	REGION READ AND INIT
	    
	    REGION Init conveyor parameters
	        
	        // Conveyor Parameter
	        // ProductionLine
	        IF #Active.Line.ProductionLine THEN
	            #ReadTransferParameters := DB_ConveyorParameters.Line.ProductionLine.Conveyor[#TransferID];
	        END_IF;
	        // EmptyLine
	        IF #Active.Line.EmptyLine THEN
	            #ReadTransferParameters := DB_ConveyorParameters.Line.EmptyLine.Conveyor[#TransferID];
	        END_IF;
	        // PackedLine
	        IF #Active.Line.PackedLine THEN
	            #ReadTransferParameters := DB_ConveyorParameters.Line.PackedLine.Conveyor[#TransferID];
	        END_IF;
	        
	    END_REGION
	    
	    REGION Sensor Filter
	        
	        // FB_Sensor
	        // called as MIDB
	        
	        #TRANSFER_SENSOR(Sensor := #ReadInputSignal.TransferSensor,
	                         SensorFilterTime := #ReadTransferParameters.SensorFilterTime,
	                         FilteredSensor => #FilteredSensor);
	        
	        // front sensor filter
	        #FRONT_SENSOR_FILTER(Sensor := #FrontSensor,
	                             SensorFilterTime := #FrontSensorFilterTime);
	        
	    END_REGION
	    
	    REGION FIRE
	        
	        // Fire signal from fire system stops the whole system
	        // System can be reset from Fire status only if the fire signal is deactivated
	        
	        // FIRE ALARM ACTIVE --> STOP SYSTEM
	        IF #ReadInputSignal.FireActive THEN
	            #StopSystemFireActive := TRUE;
	        END_IF;
	        // RESET --> FIRE ALARM
	        IF #SSR.ResetSystem AND NOT #ReadInputSignal.FireActive THEN
	            #StopSystemFireActive := FALSE;
	        END_IF;
	        
	    END_REGION
	    
	END_REGION
	
	REGION Conveyor Status
	    
	    REGION Status ON
	        
	        // ----------------------------------------->>>>>>> STATUS ON <<<<<<<-----------------------------------------
	        // FB_ConveyorStatusON
	        // called as IDMB
	        
	        #TRANSFER_STATUS_ON(SystemStartActive := #SSR.StartSystem,
	                            StatusStop := #ReadTransferStatus.Stop,
	                            StatusEStop := #ReadTransferStatus.Estop,
	                            StatusManual := #ReadTransferStatus.Manual,
	                            StatusFault := #ReadTransferStatus.Fault,
	                            FireAlarmActive := #StopSystemFireActive,
	                            StatusON => #ReadTransferStatus.ON);
	        
	    END_REGION
	    
	    REGION Status Ready
	        
	        // ----------------------------------------->>>>>>> STATUS READY <<<<<<<-----------------------------------------
	        // FB_ConveyorStatusReady
	        // called as MIDB
	        
	        #TRANSFER_STATUS_READY(StatusON := #ReadTransferStatus.ON,
	                               StatusESTOP := #ReadTransferStatus.Estop,
	                               StatusFAULT := #ReadTransferStatus.Fault,
	                               StatusMAN := #ReadTransferStatus.Manual,
	                               SignalFIRE := #StopSystemFireActive,
	                               SystemAlertTime := #ReadTransferParameters.StartUpTime,
	                               StatusReady => #ReadTransferStatus.ReadytoRun);
	        
	    END_REGION
	    
	    REGION Status Occupied
	        
	        // ----------------------------------------->>>>>>> STATUS OCCUPIED <<<<<<<-----------------------------------------
	        
	        #ReadTransferStatus.Occupied :=
	        #FilteredSensor AND
	        NOT #FRONT_SENSOR_FILTER.FilteredSensor;
	        
	    END_REGION
	    
	    REGION Status Running
	        
	        // ----------------------------------------->>>>>>> STATUS RUNNING <<<<<<<-----------------------------------------
	        
	        #ReadTransferStatus.Running := #Transfer.Command_1 OR #Transfer.Command_2;
	        
	    END_REGION
	    
	    REGION Status Fault
	        
	        // Automatic reset trigger to the needed drive after wakeup from ESTOP power miss (only if needed)
	        // will trigger for every Reset active
	        
	        #AUTO_RESET(AckIN := #SSR.ResetSystem,
	                    Ack => #AutoReset);
	        
	        // ----------------------------------------->>>>>>> STATUS FAULT <<<<<<<-----------------------------------------
	        // FC_ConveyorStatusFault
	        #TRANSFER_STATUS_FAULT(FaultActive := #ReadInputSignal.Fault,
	                               ResetFault := #SSR.ResetSystem OR #AutoReset,
	                               StatusRunning := #ReadTransferStatus.Running,
	                               FaultStatus => #ReadTransferStatus.Fault);
	        
	        #ErrorReset := #SSR.ResetSystem;
	        
	    END_REGION
	    
	    REGION Status ESTOP
	        
	        // ----------------------------------------->>>>>>> STATUS ESTOP <<<<<<<-----------------------------------------
	        
	        // EMERGENCY STOP ACTIVE --> STOP SYSTEM
	        IF #ReadInputSignal.EmergencyStop THEN
	            #ReadTransferStatus.Estop := TRUE;
	        END_IF;
	        // RESET --> EMERGENCY STOP
	        IF #AutoReset AND NOT #ReadInputSignal.EmergencyStop THEN
	            #ReadTransferStatus.Estop := FALSE;
	        END_IF;
	        
	    END_REGION
	    
	    REGION Status Manual
	        
	        // ----------------------------------------->>>>>>> STATUS MANUAL <<<<<<<-----------------------------------------
	        
	        // Write to static from IO
	        // ACTIVATE --> MANUAL MODE
	        // ProductionLine
	        IF #Active.Line.ProductionLine THEN
	            // SET --> MANUAL MODE
	            IF DB_Manual.Line.ProductionLine.Conveyor[#TransferID].ManualEnable THEN
	                #ReadTransferStatus.Manual := TRUE;
	            END_IF;
	            // RESET --> MANUAL MODE
	            IF NOT DB_Manual.Line.ProductionLine.Conveyor[#TransferID].ManualEnable AND #SSR.ResetSystem THEN
	                #ReadTransferStatus.Manual := FALSE;
	            END_IF;
	        END_IF;
	        // EmptyLine
	        IF #Active.Line.EmptyLine THEN
	            // SET --> MANUAL MODE
	            IF DB_Manual.Line.EmptyLine.Conveyor[#TransferID].ManualEnable THEN
	                #ReadTransferStatus.Manual := TRUE;
	            END_IF;
	            // RESET --> MANUAL MODE
	            IF NOT DB_Manual.Line.EmptyLine.Conveyor[#TransferID].ManualEnable AND #SSR.ResetSystem THEN
	                #ReadTransferStatus.Manual := FALSE;
	            END_IF;
	        END_IF;
	        // PackedLine
	        IF #Active.Line.PackedLine THEN
	            // SET --> MANUAL MODE
	            IF DB_Manual.Line.PackedLine.Conveyor[#TransferID].ManualEnable THEN
	                #ReadTransferStatus.Manual := TRUE;
	            END_IF;
	            // RESET --> MANUAL MODE
	            IF NOT DB_Manual.Line.PackedLine.Conveyor[#TransferID].ManualEnable AND #SSR.ResetSystem THEN
	                #ReadTransferStatus.Manual := FALSE;
	            END_IF;
	        END_IF;
	        
	    END_REGION
	    
	    REGION Status Stop
	        
	        // ----------------------------------------->>>>>>> STATUS STOP <<<<<<<-----------------------------------------
	        
	        IF #SSR.StopSystem THEN
	            #ReadTransferStatus.Stop := TRUE;
	        END_IF;
	        IF #SSR.StartSystem OR #SSR.ResetSystem THEN
	            #ReadTransferStatus.Stop := FALSE;
	        END_IF;
	        
	    END_REGION
	    
	    REGION Status Blockage
	        
	        // FB_SensorBlockage
	        // called as MIDB
	        #TRANSFER_SENSOR_BLOCKAGE(IN := #ReadTransferStatus.ReadytoRun AND #FilteredSensor AND NOT #Downstream,
	                                  PT := T#15s);
	        
	        #FRONT_SENSOR_BLOCKAGE(IN := #ReadTransferStatus.ReadytoRun AND #FrontSensor AND NOT #Downstream,
	                               PT := T#15s);
	        
	        #END_SENSOR_BLOCKAGE(IN := #ReadTransferStatus.ReadytoRun AND #EndSensor AND NOT #Downstream,
	                             PT := T#15s);
	        
	        #"LEFT/RIGHT_SENSOR_BLOCKAGE"(IN := #ReadTransferStatus.ReadytoRun AND #"Left/RightSensor" AND NOT #Downstream,
	                                      PT := T#5s);
	        
	        #ReadTransferStatus.Blockage :=
	        (#TRANSFER_SENSOR_BLOCKAGE.Q OR
	        #FRONT_SENSOR_BLOCKAGE.Q OR
	        #END_SENSOR_BLOCKAGE.Q OR
	        #"LEFT/RIGHT_SENSOR_BLOCKAGE".Q) AND
	        (#TransferDirection.Straight OR
	        #TransferDirection.toRight OR
	        #TransferDirection.toLeft);
	        
	        // ==========================
	        // Sensor Blockage: HMI Alarm
	        // ==========================
	        // Sensor blockage alarm message is written to the alarm word
	        // corresponding to the active line
	        
	        REGION alarm 
	            
	            // ==========================
	            // Sensor Blockage: HMI Alarm
	            // ==========================
	            // Sensor blockage alarm message is written to the alarm word
	            // corresponding to the active line
	            // ProductionLine
	            IF #Active.Line.ProductionLine THEN
	                DB_Alarm."word".Line.ProductionLine.Conveyor[#TransferID].%X0 := #ReadTransferStatus.Blockage;
	            END_IF;
	            // EmptyLine
	            IF #Active.Line.EmptyLine THEN
	                DB_Alarm."word".Line.EmptyLine.Conveyor[#TransferID].%X0 := #ReadTransferStatus.Blockage;
	            END_IF;
	            // PackedLine
	            IF #Active.Line.PackedLine THEN
	                DB_Alarm."word".Line.PackedLine.Conveyor[#TransferID].%X0 := #ReadTransferStatus.Blockage;
	            END_IF;
	            
	        END_REGION
	        
	    END_REGION
	    
	    REGION Visu Color
	        
	        // each and every status of the conveyor will be mentioned by different colors in HMI panel
	        
	        #VisuColor.%X8 := #ReadTransferStatus.Blockage;
	        #VisuColor.%X0 := #ReadTransferStatus.ON;
	        #VisuColor.%X1 := #ReadTransferStatus.ReadytoRun;
	        #VisuColor.%X2 := #ReadTransferStatus.Occupied;
	        #VisuColor.%X3 := #ReadTransferStatus.Running;
	        #VisuColor.%X4 := #ReadTransferStatus.Fault;
	        #VisuColor.%X5 := #ReadTransferStatus.Estop;
	        #VisuColor.%X6 := #ReadTransferStatus.Manual;
	        #VisuColor.%X7 := #ReadTransferStatus.Stop;
	        
	        // convert word to Interger value: 
	        // color will be depends on the status priority (integer value) 
	        // reference: Conveyor image in HMI screen -> property -> Apperance   
	        
	        // ProductionLine
	        IF #Active.Line.ProductionLine THEN
	            DB_VisuColor.Line.ProductionLine.Conveyor[#TransferID] :=
	            WORD_TO_INT(#VisuColor);
	        END_IF;
	        // EmptyLine
	        IF #Active.Line.EmptyLine THEN
	            DB_VisuColor.Line.EmptyLine.Conveyor[#TransferID] :=
	            WORD_TO_INT(#VisuColor);
	        END_IF;
	        // PackedLine
	        IF #Active.Line.PackedLine THEN
	            DB_VisuColor.Line.PackedLine.Conveyor[#TransferID] :=
	            WORD_TO_INT(#VisuColor);
	        END_IF;
	        
	    END_REGION
	    
	    REGION Global Status
	        
	        // write -> global status
	        // ProductionLine
	        IF #Active.Line.ProductionLine THEN
	            DB_Global.Status.Line.ProductionLine.On[#TransferID] := #ReadTransferStatus.ON;
	            DB_Global.Status.Line.ProductionLine.ReadyToRun[#TransferID] := #ReadTransferStatus.ReadytoRun;
	            DB_Global.Status.Line.ProductionLine.Occupied[#TransferID] := #ReadTransferStatus.Occupied;
	            DB_Global.Status.Line.ProductionLine.Running[#TransferID] := #ReadTransferStatus.Running;
	            DB_Global.Status.Line.ProductionLine.Fault[#TransferID] := #ReadTransferStatus.Fault;
	            DB_Global.Status.Line.ProductionLine.Estop[#TransferID] := #ReadTransferStatus.Estop;
	            DB_Global.Status.Line.ProductionLine.Manual[#TransferID] := #ReadTransferStatus.Manual;
	            DB_Global.Status.Line.ProductionLine.Stop[#TransferID] := #ReadTransferStatus.Stop;
	            DB_Global.Status.Line.ProductionLine.Blockage[#TransferID] := #ReadTransferStatus.Blockage;
	        END_IF;
	        // EmptyLine
	        IF #Active.Line.EmptyLine THEN
	            DB_Global.Status.Line.EmptyLine.On[#TransferID] := #ReadTransferStatus.ON;
	            DB_Global.Status.Line.EmptyLine.ReadyToRun[#TransferID] := #ReadTransferStatus.ReadytoRun;
	            DB_Global.Status.Line.EmptyLine.Occupied[#TransferID] := #ReadTransferStatus.Occupied;
	            DB_Global.Status.Line.EmptyLine.Running[#TransferID] := #ReadTransferStatus.Running;
	            DB_Global.Status.Line.EmptyLine.Fault[#TransferID] := #ReadTransferStatus.Fault;
	            DB_Global.Status.Line.EmptyLine.Estop[#TransferID] := #ReadTransferStatus.Estop;
	            DB_Global.Status.Line.EmptyLine.Manual[#TransferID] := #ReadTransferStatus.Manual;
	            DB_Global.Status.Line.EmptyLine.Stop[#TransferID] := #ReadTransferStatus.Stop;
	            DB_Global.Status.Line.EmptyLine.Blockage[#TransferID] := #ReadTransferStatus.Blockage;
	        END_IF;
	        // PackedLine
	        IF #Active.Line.PackedLine THEN
	            DB_Global.Status.Line.PackedLine.On[#TransferID] := #ReadTransferStatus.ON;
	            DB_Global.Status.Line.PackedLine.ReadyToRun[#TransferID] := #ReadTransferStatus.ReadytoRun;
	            DB_Global.Status.Line.PackedLine.Occupied[#TransferID] := #ReadTransferStatus.Occupied;
	            DB_Global.Status.Line.PackedLine.Running[#TransferID] := #ReadTransferStatus.Running;
	            DB_Global.Status.Line.PackedLine.Fault[#TransferID] := #ReadTransferStatus.Fault;
	            DB_Global.Status.Line.PackedLine.Estop[#TransferID] := #ReadTransferStatus.Estop;
	            DB_Global.Status.Line.PackedLine.Manual[#TransferID] := #ReadTransferStatus.Manual;
	            DB_Global.Status.Line.PackedLine.Stop[#TransferID] := #ReadTransferStatus.Stop;
	            DB_Global.Status.Line.PackedLine.Blockage[#TransferID] := #ReadTransferStatus.Blockage;
	        END_IF;
	        
	    END_REGION
	    
	END_REGION
	
	REGION Transfer Logic
	    
	    REGION infeed receive condition
	        
	        // NegEdgeUpstream
	        #NegEdgeUpstream(CLK := #Upstream);
	        
	        // item will be send into the transfer section when there is no other item
	        
	        IF #ReadTransferStatus.ReadytoRun AND
	            #Upstream AND
	            NOT #ReadTransferStatus.Occupied THEN
	            #Transfer.RcvInfeed := TRUE;
	        END_IF;
	        
	        // receive infeed tag goes to FALSE when the item from the previous conveyor is completly out of the previous conveyor
	        IF NOT #Upstream(* #NegEdgeUpstream.Q *)THEN
	            #Transfer.RcvInfeed := FALSE;
	        END_IF;
	        
	        // Receive infeed
	        #Transfer.StartSignal := #Transfer.RcvInfeed;
	        
	    END_REGION
	    
	    REGION Transfer direction outputs
	        
	        IF NOT #EndSensor AND NOT #"Left/RightSensor" AND NOT #ReadTransferStatus.Running THEN
	            
	            #sTransferDirection := #TransferDirection;
	            
	        END_IF;
	        
	        // Transfer Straight
	        
	        IF #sTransferDirection.Straight THEN
	            
	            IF #ReadTransferStatus.ReadytoRun AND
	                NOT #Transfer.RcvInfeed AND
	                #ReadTransferStatus.Occupied AND
	                NOT #Downstream
	            THEN
	                #Transfer.Command_1 := TRUE;
	                #Transfer.Command_2 := TRUE;
	            END_IF;
	            
	        END_IF;
	        
	        // Transfer Right
	        
	        IF #sTransferDirection.toRight THEN
	            
	            IF #ReadTransferStatus.ReadytoRun AND
	                NOT #Transfer.RcvInfeed AND
	                #ReadTransferStatus.Occupied AND
	                NOT #Downstream
	            THEN
	                #Transfer.Command_1 := TRUE;
	                #Transfer.Command_2 := FALSE;
	            END_IF;
	            
	        END_IF;
	        
	        // Transfer Left
	        
	        IF #sTransferDirection.toLeft THEN
	            
	            IF #ReadTransferStatus.ReadytoRun AND
	                NOT #Transfer.RcvInfeed AND
	                #ReadTransferStatus.Occupied AND
	                NOT #Downstream
	            THEN
	                #Transfer.Command_1 := FALSE;
	                #Transfer.Command_2 := TRUE;
	            END_IF;
	            
	        END_IF;
	        
	    END_REGION
	    
	    REGION TRANSFER OFF
	        
	        // Transfer commands Off
	        
	        IF NOT #ReadTransferStatus.ReadytoRun OR
	            #Transfer.RcvInfeed OR
	            (#ReadTransferStatus.Occupied AND
	            #Downstream) OR
	            NOT #ReadTransferStatus.Occupied
	        THEN
	            #Transfer.Command_1 := FALSE;
	            #Transfer.Command_2 := FALSE;
	        END_IF;
	        
	    END_REGION
	    
	    REGION Write output
	        
	        // Static to output
	        
	        #StartSignal := #Transfer.StartSignal;
	        #Cmd1 := #Transfer.Command_1;
	        #Cmd2 := #Transfer.Command_2;
	        
	    END_REGION
	    
	END_REGION
	
	
	
	
	
END_FUNCTION_BLOCK
END_NAMESPACE

NAMESPACE Global
FUNCTION_BLOCK FB_GetDiag
{ S7_Optimized_Access := 'TRUE' ; Published := 'TRUE' }
VERSION : 0.1
   VAR_INPUT 
      HardwareID : HW_ANY;
   END_VAR

   VAR_OUTPUT 
      CommunicationErrorAlarm : Bool;
   END_VAR

   VAR 
      GetDiag { S7_SetPoint := 'False'} : GetDiag;
      CheckOwnState : UInt := 5;
      CommunicationError : Bool;
   END_VAR


BEGIN
	// ==========================================================================================================================================
	// Company        : LogTech, s.r.o.
	// Created by     : Anton Vinoth Soundraraj
	// Block          : FB_GetDiag
	// Project        : LT-Lib-Block
	// ==========================================================================================================================================
	
	REGION Get_Diag
	    
	    #GetDiag.ReturnValue := GET_DIAG(MODE := #GetDiag.DiagMode,
	                                     LADDR := #HardwareID,
	                                     CNT_DIAG => #GetDiag.CountDiagDetail,
	                                     DIAG := #GetDiag.MyDiag);
	END_REGION
	
	REGION Communiation_Error
	    
	    IF #GetDiag.MyDiag.OwnState = #CheckOwnState THEN
	        #CommunicationErrorAlarm := TRUE;
	    ELSE
	        #CommunicationErrorAlarm := FALSE;
	    END_IF;
	    
	    IF #GetDiag.MyDiag.OwnState = #CheckOwnState THEN
	        #CommunicationError := TRUE;
	    ELSE
	        #CommunicationError := FALSE;
	    END_IF;
	    
	END_REGION
	
	
END_FUNCTION_BLOCK
END_NAMESPACE

NAMESPACE Global
FUNCTION_BLOCK FB_HardwareDiag
{ S7_Optimized_Access := 'TRUE' ; Published := 'TRUE' }
VERSION : 0.1
   VAR 
      "BW-ASi -10.106.129.143" { S7_SetPoint := 'False'} : FB_GetDiag;
      "BW-ASi -10.106.129.200" : FB_GetDiag;
      "Cognex -10.106.129.24" { S7_SetPoint := 'False'} : FB_GetDiag;
      "Cognex -10.106.129.25" : FB_GetDiag;
      "Cognex -10.106.129.26" : FB_GetDiag;
      "Cognex -10.106.129.27" : FB_GetDiag;
      "IMC - 10.106.129.84" : FB_GetDiag;
      "IMC - 10.106.129.85" : FB_GetDiag;
      "IMC - 10.106.129.86" : FB_GetDiag;
      "IMC - 10.106.129.87" : FB_GetDiag;
      "IMC - 10.106.129.88" : FB_GetDiag;
   END_VAR


BEGIN
	// ==========================================================================================================================================
	// Company        : LogTech, s.r.o.
	// Created by     : Anton Vinoth Soundraraj
	// Block          : FB_HardwareDiag
	// Project        : Lékarna DC Chrudim
	// Project number : 23-157
	// ==========================================================================================================================================
	
	
	REGION BW ASi module
	    
	    
	    #"BW-ASi -10.106.129.143"(CommunicationErrorAlarm=> DB_Alarm.CommunicationFault."BW-ASi".%X0);  // remove for simulation testing HardwareID:= _."ASi-GW~IODevice",
	    
	    #"BW-ASi -10.106.129.200"(CommunicationErrorAlarm=> DB_Alarm.CommunicationFault."BW-ASi".%X1);
	    
	END_REGION
	
	
	REGION Cognex
	    
	    #"Cognex -10.106.129.24"(CommunicationErrorAlarm=> DB_Alarm.CommunicationFault.Cognex.%X0);
	    
	    
	    #"Cognex -10.106.129.25"(CommunicationErrorAlarm=> DB_Alarm.CommunicationFault.Cognex.%X1);
	    
	    
	    #"Cognex -10.106.129.26"(CommunicationErrorAlarm=> DB_Alarm.CommunicationFault.Cognex.%X2);
	    
	    
	    #"Cognex -10.106.129.27"(CommunicationErrorAlarm=> DB_Alarm.CommunicationFault.Cognex.%X3);
	    
	    
	END_REGION
	
	REGION IMC
	    
	    #"IMC - 10.106.129.84"(CommunicationErrorAlarm=>DB_Alarm.CommunicationFault.IMC.%X0);
	    
	    #"IMC - 10.106.129.85"(CommunicationErrorAlarm=>DB_Alarm.CommunicationFault.IMC.%X1);
	    
	    #"IMC - 10.106.129.86"(CommunicationErrorAlarm=>DB_Alarm.CommunicationFault.IMC.%X1);
	    
	    #"IMC - 10.106.129.87"(CommunicationErrorAlarm=>DB_Alarm.CommunicationFault.IMC.%X2);
	    
	    #"IMC - 10.106.129.88"(CommunicationErrorAlarm=>DB_Alarm.CommunicationFault.IMC.%X3);
	    
	END_REGION
	
	
	
	
	
	
	
END_FUNCTION_BLOCK
END_NAMESPACE

NAMESPACE Global
FUNCTION_BLOCK FB_VisuAlarm
{ S7_Optimized_Access := 'TRUE' ; Published := 'TRUE' }
VERSION : 0.1
   VAR 
      noAlarmState : Bool;
      CommunicationFault : Struct
         PLC : Word;
         "BW-ASi" : Word;
         Cognex : Word;
         Mabs : Word;
      END_STRUCT;
      "BW-ASi" : Struct
         "BW_ASi143 -MCC100 -210KE3 -ConfigErr_Circuit1_Slave(0-15)A_1" : Word;
         "BW_ASi143 -MCC100 -210KE3 -ConfigErr_Circuit1_Slave(16-31)A" : Word;
         "BW_ASi143 -MCC100 -210KE3 -ConfigErr_Circuit1_Slave(0-15)B_1" : Word;
         "BW_ASi143 -MCC100 -210KE3 -ConfigErr_Circuit1_Slave(16-31)B" : Word;
         "BW_ASi143 -MCC100 -210KE3 -PeriErr_Circuit1_Slave(0-15)A_1" : Word;
         "BW_ASi143 -MCC100 -210KE3 -PeriErr_Circuit1_Slave(16-31)A" : Word;
         "BW_ASi143 -MCC100 -210KE3 -PeriErr_Circuit1_Slave(0-15)B_1" : Word;
         "BW_ASi143 -MCC100 -210KE3 -PeriErr_Circuit1_Slave(16-31)B" : Word;
         "BW_ASi143 -MCC100 -210KE3 -ConfigErr_Circuit2_Slave(0-15)A" : Word;
         "BW_ASi143 -MCC100 -210KE3 -ConfigErr_Circuit2_Slave(16-31)A" : Word;
         "BW_ASi143 -MCC100 -210KE3 -ConfigErr_Circuit2_Slave(0-15)B" : Word;
         "BW_ASi143 -MCC100 -210KE3 -ConfigErr_Circuit2_Slave(16-31)B" : Word;
         "BW_ASi143 -MCC100 -210KE3 -PeriErr_Circuit2_Slave(0-15)A" : Word;
         "BW_ASi143 -MCC100 -210KE3 -PeriErr_Circuit2_Slave(16-31)A" : Word;
         "BW_ASi143 -MCC100 -210KE3 -PeriErr_Circuit2_Slave(0-15)B" : Word;
         "BW_ASi143 -MCC100 -210KE3 -PeriErr_Circuit2_Slave(16-31)B" : Word;
         "BW_ASi200 -MCC300 -210KE3 -ConfigErr_Circuit1_Slave(0-15)A" : Word;
         "BW_ASi200 -MCC300 -210KE3 -ConfigErr_Circuit1_Slave(16-31)A" : Word;
         "BW_ASi200 -MCC300 -210KE3 -ConfigErr_Circuit1_Slave(0-15)B" : Word;
         "BW_ASi200 -MCC300 -210KE3 -ConfigErr_Circuit1_Slave(16-31)B" : Word;
         "BW_ASi200 -MCC300 -210KE3 -PeriErr_Circuit1_Slave(0-15)A" : Word;
         "BW_ASi200 -MCC300 -210KE3 -PeriErr_Circuit1_Slave(16-31)A" : Word;
         "BW_ASi200 -MCC300 -210KE3 -PeriErr_Circuit1_Slave(0-15)B" : Word;
         "BW_ASi200 -MCC300 -210KE3 -PeriErr_Circuit1_Slave(16-31)B" : Word;
         "BW_ASi200 -MCC300 -210KE3 -ConfigErr_Circuit2_Slave(0-15)A" : Word;
         "BW_ASi200 -MCC300 -210KE3 -ConfigErr_Circuit2_Slave(16-31)A" : Word;
         "BW_ASi200 -MCC300 -210KE3 -ConfigErr_Circuit2_Slave(0-15)B" : Word;
         "BW_ASi200 -MCC300 -210KE3 -ConfigErr_Circuit2_Slave(16-31)B" : Word;
         "BW_ASi200 -MCC300 -210KE3 -PeriErr_Circuit2_Slave(0-15)A" : Word;
         "BW_ASi200 -MCC300 -210KE3 -PeriErr_Circuit2_Slave(16-31)A" : Word;
         "BW_ASi200 -MCC300 -210KE3 -PeriErr_Circuit2_Slave(0-15)B" : Word;
         "BW_ASi200 -MCC300 -210KE3 -PeriErr_Circuit2_Slave(16-31)B" : Word;
      END_STRUCT;
      "word" : Struct
         Line : Struct
            ProductionLine : Struct
               Conveyor : Array[_.gminProductionLine.._.gmaxProductionLine] of Word;
            END_STRUCT;
            EmptyLine : Struct
               Conveyor : Array[_.gminEmptyLine.._.gmaxEmptyLine] of Word;
            END_STRUCT;
            PackedLine : Struct
               Conveyor : Array[_.gminPackedLine.._.gmaxPackedLine] of Word;
            END_STRUCT;
         END_STRUCT;
      END_STRUCT;
   END_VAR


BEGIN
	// ==========================================================================================================================================
	// Company        : LogTech, s.r.o.
	// Created by     : Mahmoud Elnady
	// Block          : FC_VisuAlarm
	// Project        : Lékárna Chrudim
	// Project number : 23-157
	// ==========================================================================================================================================
	REGION initial state
	    
	    // ESTOP alarm has priority
	    // So, if there are any estop active, other alarms can't be displayed on Alarm screen
	    
	    // no alarm state
	    #noAlarmState :=
	    IDB_GlobalStatus.Line.ProductionLine.Estop OR
	    IDB_GlobalStatus.Line.ProductionLine.Estop OR
	    IDB_GlobalStatus.Line.ProductionLine.Estop;
	    
	    IF #noAlarmState THEN
	        
	        DB_Alarm."BW-ASi" := #"BW-ASi";
	        DB_Alarm.CommunicationFault := #CommunicationFault;
	        DB_Alarm."word" := #word;
	        //"DB_Alarm".CircuitBreaker := #CircuitBreaker;
	        
	    END_IF;
	    
	END_REGION
	
	REGION ASi Config and Peri alarm
	    
	    IF NOT #noAlarmState THEN
	        // ASi gateway: MCC100-bw23: Circuit 1
	        DB_Alarm."BW-ASi"."BW_ASi143 -MCC100 -210KE3 -ConfigErr_Circuit1_Slave(0-15)A" := _."BW_ASi143 -MCC100 -210KE3 -ConfigErr_Circuit1_Slave(0-15)A";
	        DB_Alarm."BW-ASi"."BW_ASi143 -MCC100 -210KE3 -ConfigErr_Circuit1_Slave(16-31)A" := _."BW_ASi143 -MCC100 -210KE3 -ConfigErr_Circuit1_Slave(16-31)A";
	        DB_Alarm."BW-ASi"."BW_ASi143 -MCC100 -210KE3 -ConfigErr_Circuit1_Slave(0-15)B" := _."BW_ASi143 -MCC100 -210KE3 -ConfigErr_Circuit1_Slave(0-15)B";
	        DB_Alarm."BW-ASi"."BW_ASi143 -MCC100 -210KE3 -ConfigErr_Circuit1_Slave(16-31)B" := _."BW_ASi143 -MCC100 -210KE3 -ConfigErr_Circuit1_Slave(16-31)B";
	        DB_Alarm."BW-ASi"."BW_ASi143 -MCC100 -210KE3 -PeriErr_Circuit1_Slave(0-15)A" := _."BW_ASi143 -MCC100 -210KE3 -PeriErr_Circuit1_Slave(0-15)A";
	        DB_Alarm."BW-ASi"."BW_ASi143 -MCC100 -210KE3 -PeriErr_Circuit1_Slave(16-31)A" := _."BW_ASi143 -MCC100 -210KE3 -PeriErr_Circuit1_Slave(16-31)A";
	        DB_Alarm."BW-ASi"."BW_ASi143 -MCC100 -210KE3 -PeriErr_Circuit1_Slave(0-15)B" := _."BW_ASi143 -MCC100 -210KE3 -PeriErr_Circuit1_Slave(0-15)B";
	        DB_Alarm."BW-ASi"."BW_ASi143 -MCC100 -210KE3 -PeriErr_Circuit1_Slave(16-31)B" := _."BW_ASi143 -MCC100 -210KE3 -PeriErr_Circuit1_Slave(16-31)B";
	        // ASi gateway: MCC100-bw23: Circuit 2
	        DB_Alarm."BW-ASi"."BW_ASi143 -MCC100 -210KE3 -ConfigErr_Circuit1_Slave(0-15)A" := _."BW_ASi143 -MCC100 -210KE3 -ConfigErr_Circuit1_Slave(0-15)A";
	        DB_Alarm."BW-ASi"."BW_ASi143 -MCC100 -210KE3 -ConfigErr_Circuit1_Slave(16-31)A" := _."BW_ASi143 -MCC100 -210KE3 -ConfigErr_Circuit1_Slave(16-31)A";
	        DB_Alarm."BW-ASi"."BW_ASi143 -MCC100 -210KE3 -ConfigErr_Circuit1_Slave(0-15)B" := _."BW_ASi143 -MCC100 -210KE3 -ConfigErr_Circuit1_Slave(0-15)B";
	        DB_Alarm."BW-ASi"."BW_ASi143 -MCC100 -210KE3 -ConfigErr_Circuit1_Slave(16-31)B" := _."BW_ASi143 -MCC100 -210KE3 -ConfigErr_Circuit1_Slave(16-31)B";
	        DB_Alarm."BW-ASi"."BW_ASi143 -MCC100 -210KE3 -PeriErr_Circuit1_Slave(0-15)A" := _."BW_ASi143 -MCC100 -210KE3 -PeriErr_Circuit1_Slave(0-15)A";
	        DB_Alarm."BW-ASi"."BW_ASi143 -MCC100 -210KE3 -PeriErr_Circuit1_Slave(16-31)A" := _."BW_ASi143 -MCC100 -210KE3 -PeriErr_Circuit1_Slave(16-31)A";
	        DB_Alarm."BW-ASi"."BW_ASi143 -MCC100 -210KE3 -PeriErr_Circuit1_Slave(0-15)B" := _."BW_ASi143 -MCC100 -210KE3 -PeriErr_Circuit1_Slave(0-15)B";
	        DB_Alarm."BW-ASi"."BW_ASi143 -MCC100 -210KE3 -PeriErr_Circuit1_Slave(16-31)B" := _."BW_ASi143 -MCC100 -210KE3 -PeriErr_Circuit1_Slave(16-31)B";
	        // ASi gateway: MCC300-bw31 : Circuit 1
	        DB_Alarm."BW-ASi"."BW_ASi200 -MCC300 -210KE3 -ConfigErr_Circuit1_Slave(0-15)A" := _."BW_ASi200 -MCC300 -210KE3 -ConfigErr_Circuit1_Slave(0-15)A";
	        DB_Alarm."BW-ASi"."BW_ASi200 -MCC300 -210KE3 -ConfigErr_Circuit1_Slave(16-31)A" := _."BW_ASi200 -MCC300 -210KE3 -ConfigErr_Circuit1_Slave(16-31)A";
	        DB_Alarm."BW-ASi"."BW_ASi200 -MCC300 -210KE3 -ConfigErr_Circuit1_Slave(0-15)B" := _."BW_ASi200 -MCC300 -210KE3 -ConfigErr_Circuit1_Slave(0-15)B";
	        DB_Alarm."BW-ASi"."BW_ASi200 -MCC300 -210KE3 -ConfigErr_Circuit1_Slave(16-31)B" := _."BW_ASi200 -MCC300 -210KE3 -ConfigErr_Circuit1_Slave(16-31)B";
	        DB_Alarm."BW-ASi"."BW_ASi200 -MCC300 -210KE3 -PeriErr_Circuit1_Slave(0-15)A" := _."BW_ASi200 -MCC300 -210KE3 -PeriErr_Circuit1_Slave(0-15)A";
	        DB_Alarm."BW-ASi"."BW_ASi200 -MCC300 -210KE3 -PeriErr_Circuit1_Slave(16-31)A" := _."BW_ASi200 -MCC300 -210KE3 -PeriErr_Circuit1_Slave(16-31)A";
	        DB_Alarm."BW-ASi"."BW_ASi200 -MCC300 -210KE3 -PeriErr_Circuit1_Slave(0-15)B" := _."BW_ASi200 -MCC300 -210KE3 -PeriErr_Circuit1_Slave(0-15)B";
	        DB_Alarm."BW-ASi"."BW_ASi200 -MCC300 -210KE3 -PeriErr_Circuit1_Slave(16-31)B" := _."BW_ASi200 -MCC300 -210KE3 -PeriErr_Circuit1_Slave(16-31)B";
	        // ASi gateway: MCC300-bw31 : Circuit 2
	        DB_Alarm."BW-ASi"."BW_ASi200 -MCC300 -210KE3 -ConfigErr_Circuit2_Slave(0-15)A" := _."BW_ASi200 -MCC300 -210KE3 -ConfigErr_Circuit2_Slave(0-15)A";
	        DB_Alarm."BW-ASi"."BW_ASi200 -MCC300 -210KE3 -ConfigErr_Circuit2_Slave(16-31)A" := _."BW_ASi200 -MCC300 -210KE3 -ConfigErr_Circuit2_Slave(16-31)A";
	        DB_Alarm."BW-ASi"."BW_ASi200 -MCC300 -210KE3 -ConfigErr_Circuit2_Slave(0-15)B" := _."BW_ASi200 -MCC300 -210KE3 -ConfigErr_Circuit2_Slave(0-15)B";
	        DB_Alarm."BW-ASi"."BW_ASi200 -MCC300 -210KE3 -ConfigErr_Circuit2_Slave(16-31)B" := _."BW_ASi200 -MCC300 -210KE3 -ConfigErr_Circuit2_Slave(16-31)B";
	        DB_Alarm."BW-ASi"."BW_ASi200 -MCC300 -210KE3 -PeriErr_Circuit2_Slave(0-15)A" := _."BW_ASi200 -MCC300 -210KE3 -PeriErr_Circuit2_Slave(0-15)A";
	        DB_Alarm."BW-ASi"."BW_ASi200 -MCC300 -210KE3 -PeriErr_Circuit2_Slave(16-31)A" := _."BW_ASi200 -MCC300 -210KE3 -PeriErr_Circuit2_Slave(16-31)A";
	        DB_Alarm."BW-ASi"."BW_ASi200 -MCC300 -210KE3 -PeriErr_Circuit2_Slave(0-15)B" := _."BW_ASi200 -MCC300 -210KE3 -PeriErr_Circuit2_Slave(0-15)B";
	        DB_Alarm."BW-ASi"."BW_ASi200 -MCC300 -210KE3 -PeriErr_Circuit2_Slave(16-31)B" := _."BW_ASi200 -MCC300 -210KE3 -PeriErr_Circuit2_Slave(16-31)B";
	    ELSE
	        // ASi gateway: MCC100-bw23: Circuit 1
	        DB_Alarm."BW-ASi"."BW_ASi143 -MCC100 -210KE3 -ConfigErr_Circuit1_Slave(0-15)A" := 0;
	        DB_Alarm."BW-ASi"."BW_ASi143 -MCC100 -210KE3 -ConfigErr_Circuit1_Slave(16-31)A" := 0;
	        DB_Alarm."BW-ASi"."BW_ASi143 -MCC100 -210KE3 -ConfigErr_Circuit1_Slave(0-15)B" := 0;
	        DB_Alarm."BW-ASi"."BW_ASi143 -MCC100 -210KE3 -ConfigErr_Circuit1_Slave(16-31)B" := 0;
	        DB_Alarm."BW-ASi"."BW_ASi143 -MCC100 -210KE3 -PeriErr_Circuit1_Slave(0-15)A" := 0;
	        DB_Alarm."BW-ASi"."BW_ASi143 -MCC100 -210KE3 -PeriErr_Circuit1_Slave(16-31)A" := 0;
	        DB_Alarm."BW-ASi"."BW_ASi143 -MCC100 -210KE3 -PeriErr_Circuit1_Slave(0-15)B" := 0;
	        DB_Alarm."BW-ASi"."BW_ASi143 -MCC100 -210KE3 -PeriErr_Circuit1_Slave(16-31)B" := 0;
	        // ASi gateway: MCC100-bw23: Circuit 2
	        DB_Alarm."BW-ASi"."BW_ASi143 -MCC100 -210KE3 -ConfigErr_Circuit1_Slave(0-15)A" := 0;
	        DB_Alarm."BW-ASi"."BW_ASi143 -MCC100 -210KE3 -ConfigErr_Circuit1_Slave(16-31)A" := 0;
	        DB_Alarm."BW-ASi"."BW_ASi143 -MCC100 -210KE3 -ConfigErr_Circuit1_Slave(0-15)B" := 0;
	        DB_Alarm."BW-ASi"."BW_ASi143 -MCC100 -210KE3 -ConfigErr_Circuit1_Slave(16-31)B" := 0;
	        DB_Alarm."BW-ASi"."BW_ASi143 -MCC100 -210KE3 -PeriErr_Circuit1_Slave(0-15)A" := 0;
	        DB_Alarm."BW-ASi"."BW_ASi143 -MCC100 -210KE3 -PeriErr_Circuit1_Slave(16-31)A" := 0;
	        DB_Alarm."BW-ASi"."BW_ASi143 -MCC100 -210KE3 -PeriErr_Circuit1_Slave(0-15)B" := 0;
	        DB_Alarm."BW-ASi"."BW_ASi143 -MCC100 -210KE3 -PeriErr_Circuit1_Slave(16-31)B" := 0;
	        // ASi gateway: MCC300-bw31 : Circuit 1
	        DB_Alarm."BW-ASi"."BW_ASi200 -MCC300 -210KE3 -ConfigErr_Circuit1_Slave(0-15)A" := 0;
	        DB_Alarm."BW-ASi"."BW_ASi200 -MCC300 -210KE3 -ConfigErr_Circuit1_Slave(16-31)A" := 0;
	        DB_Alarm."BW-ASi"."BW_ASi200 -MCC300 -210KE3 -ConfigErr_Circuit1_Slave(0-15)B" := 0;
	        DB_Alarm."BW-ASi"."BW_ASi200 -MCC300 -210KE3 -ConfigErr_Circuit1_Slave(16-31)B" := 0;
	        DB_Alarm."BW-ASi"."BW_ASi200 -MCC300 -210KE3 -PeriErr_Circuit1_Slave(0-15)A" := 0;
	        DB_Alarm."BW-ASi"."BW_ASi200 -MCC300 -210KE3 -PeriErr_Circuit1_Slave(16-31)A" := 0;
	        DB_Alarm."BW-ASi"."BW_ASi200 -MCC300 -210KE3 -PeriErr_Circuit1_Slave(0-15)B" := 0;
	        DB_Alarm."BW-ASi"."BW_ASi200 -MCC300 -210KE3 -PeriErr_Circuit1_Slave(16-31)B" := 0;
	        // ASi gateway: MCC300-bw31 : Circuit 2
	        DB_Alarm."BW-ASi"."BW_ASi200 -MCC300 -210KE3 -ConfigErr_Circuit2_Slave(0-15)A" := 0;
	        DB_Alarm."BW-ASi"."BW_ASi200 -MCC300 -210KE3 -ConfigErr_Circuit2_Slave(16-31)A" := 0;
	        DB_Alarm."BW-ASi"."BW_ASi200 -MCC300 -210KE3 -ConfigErr_Circuit2_Slave(0-15)B" := 0;
	        DB_Alarm."BW-ASi"."BW_ASi200 -MCC300 -210KE3 -ConfigErr_Circuit2_Slave(16-31)B" := 0;
	        DB_Alarm."BW-ASi"."BW_ASi200 -MCC300 -210KE3 -PeriErr_Circuit2_Slave(0-15)A" := 0;
	        DB_Alarm."BW-ASi"."BW_ASi200 -MCC300 -210KE3 -PeriErr_Circuit2_Slave(16-31)A" := 0;
	        DB_Alarm."BW-ASi"."BW_ASi200 -MCC300 -210KE3 -PeriErr_Circuit2_Slave(0-15)B" := 0;
	        DB_Alarm."BW-ASi"."BW_ASi200 -MCC300 -210KE3 -PeriErr_Circuit2_Slave(16-31)B" := 0;
	        
	    END_IF;
	    
	END_REGION
	
	
END_FUNCTION_BLOCK
END_NAMESPACE

NAMESPACE Global
FUNCTION FC_SafetyAlarm : Void
{ S7_Optimized_Access := 'TRUE' ; Published := 'FALSE' }
VERSION : 0.1

BEGIN
	// ==========================================================================================================================================
	// Company        : LogTech, s.r.o.
	// Created by     : Mahmoud Elnady
	// Block          : FB_Main_LineA1
	// Project        : Lékárna Chrudim
	// Project number : 23-157
	// ==========================================================================================================================================
	
	REGION HMI Alarm
	    
	    DB_Alarm.Estop.%X0 :=
	    _.DB_SafetyStandard.PressReset;
	    DB_Alarm.Estop.%X1 :=
	    _.DB_SafetyStandard.ToStandard.EstopActive;
	    DB_Alarm.Estop.%X2 :=
	    _.DB_SafetyStandard.ToHMI."PhaseOK -MCC001";    
	    DB_Alarm.Estop.%X3 :=
	    _.DB_SafetyStandard.ToHMI."EstopPB -MCC001+MCC001-SF1";
	    
	END_REGION
END_FUNCTION
END_NAMESPACE

NAMESPACE EmptyLine
FUNCTION_BLOCK FB_Merging
{ S7_Optimized_Access := 'TRUE' ; Published := 'TRUE' }
VERSION : 0.1
   VAR 
      "Merge_J1.2.4" : _.Global.FB_Merging;
   END_VAR

   VAR_TEMP 
      Priority : Struct
         Straight : Bool;
         Arm : Bool;
      END_STRUCT;
   END_VAR


BEGIN
	// ==========================================================================================================================================
	// Company        : LogTech, s.r.o.
	// Created by     : Anton Vinoth Soundraraj
	// Block          : FB_Merging
	// Project        : Lékarna DC Chrudim
	// Project number : 23-157
	// ==========================================================================================================================================
	
	
	#"Merge_J1.2.4"(StraightSensor := IDB_EmptyLine."J1.2.3".FilteredSensor,
	                ArmSensor      := IDB_EmptyLine."J2.4.1".FilteredSensor);
	
	
	
END_FUNCTION_BLOCK
END_NAMESPACE

NAMESPACE EmptyLine
FUNCTION_BLOCK FB_ToggleDir
{ S7_Optimized_Access := 'TRUE' ; Published := 'FALSE' }
VERSION : 0.1
   VAR 
      "J1.5.4" : _.Global.ToggelDir;
      "Toggle_J1.5.4" : Struct
         StarightDir : Bool;
         ArmDir : Bool;
      END_STRUCT;
   END_VAR


BEGIN
	// ==========================================================================================================================================
	// Company        : LogTech, s.r.o.
	// Created by     : Mahmoud Elnady
	// Block          : FB_Toggel Direction
	// Project        : Lekarna, Chrudim -PLC001 -MCC001
	// Project number : 23-157
	// ==========================================================================================================================================
	
	REGION J1.5.4
	    REGION J1.5.4
	        #"J1.5.4"(Sensor := IDB_EmptyLine."J1.5.4".FilteredSensor,
	                  ArmSensor := IDB_EmptyLine."K1.1.1".FilteredSensor,
	                  StraightSensor :=  IDB_EmptyLine."J1.7.1".FilteredSensor,
	                  Toggle => #"Toggle_J1.5.4");
	    END_REGION
	    
	    REGION Straight
	        // Go Straight
	        IF #"Toggle_J1.5.4".StarightDir THEN
	            // Statement section IF
	            ToteDir.Conveyor[_."J1.6.1"].Straight := TRUE;
	            ToteDir.Conveyor[_."J1.6.1"].toRight := FALSE;
	            ToteDir.Conveyor[_."J1.6.1"].toLeft := FALSE;
	        END_IF;
	    END_REGION
	    
	    
	    REGION GoToLeft
	        //Go to the left
	        IF #"Toggle_J1.5.4".ArmDir THEN
	            // Statement section IF
	            ToteDir.Conveyor[_."J1.6.1"].Straight := FALSE;
	            ToteDir.Conveyor[_."J1.6.1"].toRight := FALSE;
	            ToteDir.Conveyor[_."J1.6.1"].toLeft := TRUE;
	        END_IF;
	    END_REGION
	END_REGION
	
	
	
END_FUNCTION_BLOCK
END_NAMESPACE

NAMESPACE Global
FUNCTION_BLOCK ToggelDir
{ S7_Optimized_Access := 'TRUE' ; Published := 'TRUE' }
VERSION : 0.1
   VAR_INPUT 
      Sensor : Bool;
      ArmSensor : Bool;
      StraightSensor : Bool;
   END_VAR

   VAR_OUTPUT 
      Toggle : Struct
         StarightDirection : Bool;
         ArmDirection : Bool;
      END_STRUCT;
   END_VAR

   VAR 
      UpCounter {InstructionName := 'CTU_INT'; LibVersion := '1.0'; S7_SetPoint := 'False'} : CTU_INT;
   END_VAR
   VAR RETAIN
      statResetCounter { S7_SetPoint := 'True'} : Bool;
   END_VAR
   VAR 
      SortAll : Struct
         Staright : Bool;
         Arm : Bool;
      END_STRUCT;
   END_VAR


BEGIN
	// ==========================================================================================================================================
	// Company        : LogTech, s.r.o.
	// Created by     : Mahmoud Elnady
	// Block          : FB_Toggel Direction
	// Project        : Lekarna, Chrudim -PLC001 -MCC001
	// Project number : 23-157
	// ==========================================================================================================================================
	
	// =============================
	// REGION Counter
	// Toggle counter: 0 = Straight, 1 = Arm
	// =============================
	IF #UpCounter.CV >= #UpCounter.PV THEN
	    #statResetCounter := TRUE;
	ELSE
	    #statResetCounter := FALSE;
	END_IF;
	
	#UpCounter(
	           CU := #Sensor,          // input pulse to count
	           R := #statResetCounter, // reset when PV reached
	           PV := 2                 // count up to 2 (0 → 1 → reset)
	);
	
	// =============================
	// REGION SortAll
	// Detect which sensor requests sorting
	// =============================
	#SortAll.Staright := #StraightSensor AND NOT #ArmSensor;
	#SortAll.Arm := #ArmSensor AND NOT #StraightSensor;
	
	// =============================
	// REGION Direction Selection
	// Decide final direction without contradiction
	// =============================
	IF #SortAll.Staright THEN
	    // Straight has priority if its sensor is active
	    #Toggle.StarightDirection := TRUE;
	    #Toggle.ArmDirection := FALSE;
	    
	ELSIF #SortAll.Arm THEN
	    // Arm if its sensor is active
	    #Toggle.StarightDirection := FALSE;
	    #Toggle.ArmDirection := TRUE;
	    
	ELSE
	    // No sensors → fall back to counter toggle
	    IF #UpCounter.CV = 0 THEN
	        #Toggle.StarightDirection := TRUE;
	        #Toggle.ArmDirection := FALSE;
	    ELSE // CV = 1
	        #Toggle.StarightDirection := FALSE;
	        #Toggle.ArmDirection := TRUE;
	    END_IF;
	END_IF;
	
	
	
	
	
	
	
	    
	    
	
	
	
END_FUNCTION_BLOCK
END_NAMESPACE

NAMESPACE Global
FUNCTION_BLOCK FB_EnergySave
{ S7_Optimized_Access := 'TRUE' ; Published := 'TRUE' }
VERSION : 0.1
   VAR_INPUT 
      StatusReady : Bool;
      StatusOccupied : Bool;
      StartUpIN : Bool;
      USOcc : Bool;
      EnergySaveTimePT : Time;
   END_VAR

   VAR_OUTPUT 
      EnergySaveTimeET : Time;
      EnergySaveOut : Bool;
   END_VAR

   VAR 
      EnergySaveTimer {InstructionName := 'IEC_TIMER'; LibVersion := '1.0'} : IEC_TIMER;
      EnergySave { S7_SetPoint := 'True'} : Bool;
   END_VAR


BEGIN
	// ==========================================================================================================================================================================================
	// Company       : LogTech, s.r.o.
	// Created by    : Anton Vinoth Soundraraj
	// Block         : FB_EnergySave
	// Project       : LT-Lib-Block
	// ==========================================================================================================================================================================================
	
	REGION Energy Save
	    
	    // Start energy save timer under certain conditions
	    #EnergySave := NOT #StatusReady OR #StatusOccupied OR #USOcc OR #StartUpIN;
	    
	    // Conveyor running under energy save condition for the preset time which is according to the length of the conveyor
	    #EnergySaveTimer.TOF(IN := #EnergySave,
	                         PT := #EnergySaveTimePT,
	                         Q => #EnergySaveOut,
	                         ET => #EnergySaveTimeET);
	    
	END_REGION
END_FUNCTION_BLOCK
END_NAMESPACE

NAMESPACE Global
FUNCTION_BLOCK FB_RunStop
{ S7_Optimized_Access := 'TRUE' ; Published := 'TRUE' }
VERSION : 0.1
   VAR_INPUT 
      StatusReady : Bool;
      StatusOccu : Bool;
      MotorReverseIN : Bool;
      DSOcc : Bool;
      USOcc : Bool;
      EnergySave : Bool;
      ILStop : Bool;
      PecBlockage : Bool;
   END_VAR

   VAR_OUTPUT 
      MotorForward : Bool;
      MotorReverse : Bool;
   END_VAR

   VAR 
      RunRevIN : Bool;
      RunRev : Bool;
      RunFor : Bool;
   END_VAR


BEGIN
	// ==========================================================================================================================================================================
	// Company       : LogTech, s.r.o.
	// Created by    : Anton Vinoth Soundraraj
	// Block         : FB_RunStop
	// Project       : LT-Lib-Block
	// ==========================================================================================================================================================================
	
	REGION Run/Stop Forward
	    
	    // Run forward
	    #RunFor := #StatusReady AND NOT #MotorReverseIN AND
	    ((#StatusOccu AND NOT #DSOcc) OR (NOT #StatusOccu AND #USOcc)
	    OR #EnergySave) AND NOT #PecBlockage;
	    
	    // Stop forward
	    IF NOT #StatusReady
	        OR (#StatusOccu AND #DSOcc)
	        OR #ILStop OR NOT #EnergySave OR #MotorReverseIN
	        OR #PecBlockage
	    THEN
	        #RunFor := FALSE;
	    END_IF;
	    
	    #MotorForward := #RunFor;
	    
	END_REGION
	
	REGION Run/Stop Reverse
	    
	    // Run reverse 
	    #RunRevIN := #MotorReverseIN;
	    #RunRev := #StatusReady AND #RunRevIN AND NOT #RunFor;
	    
	    // Stop reverse
	    IF NOT #StatusReady AND NOT #RunRevIN THEN
	        #RunRev := FALSE;
	    END_IF;
	    
	    #MotorReverse := #RunRev;
	    
	END_REGION
END_FUNCTION_BLOCK
END_NAMESPACE

NAMESPACE Global
FUNCTION_BLOCK FB_Sensor
{ S7_Optimized_Access := 'TRUE' ; Published := 'TRUE' }
VERSION : 0.1
   VAR_INPUT 
      Sensor : Bool;
      SensorFilterTime : Array[1..2] of Time;   // Filtering time
   END_VAR

   VAR_OUTPUT 
      FilteredSensor : Bool;
   END_VAR

   VAR 
      SensorFilterTimer {InstructionName := 'IEC_TIMER'; LibVersion := '1.0'} : Array[1..2] of IEC_TIMER;
      Filtering : Struct
         Sensor : Bool;
      END_STRUCT;
      Filtered : Struct
         Sensor : Bool;
      END_STRUCT;
      SensorEdge : Struct
         Positive : Bool;
         Negative : Bool;
      END_STRUCT;
      PosEdge {InstructionName := 'R_TRIG'; LibVersion := '1.0'; S7_SetPoint := 'False'} : R_TRIG;
      NegEdge {InstructionName := 'F_TRIG'; LibVersion := '1.0'} : F_TRIG;
   END_VAR


BEGIN
	// ==========================================================================================================================================================================
	// Company       : LogTech, s.r.o.
	// Created by    : Anton Vinoth Soundraraj
	// Block         : FB_Sensor
	// Project       : LT-Lib-Block
	// ==========================================================================================================================================================================
	
	REGION Sensor Filter
	    
	    // Filter timer 1 sending the sensor active signal to the process after preset time
	    #SensorFilterTimer[1].TON(IN := #Sensor,
	                              PT := #SensorFilterTime[1],
	                              Q => #Filtering.Sensor);
	    
	    // Filter timer 2 stop the sensor active signal from the process after preset time
	    #SensorFilterTimer[2].TOF(IN := #Filtering.Sensor,
	                              PT := #SensorFilterTime[2],
	                              Q => #Filtered.Sensor);
	    
	    // Static to output
	    #FilteredSensor := #Filtered.Sensor;
	    
	END_REGION
	
	REGION Sensor Edge Detection
	    
	    #PosEdge(CLK := #Filtered.Sensor);
	    #NegEdge(CLK := #Sensor);
	    #SensorEdge.Positive := #PosEdge.Q;
	    #SensorEdge.Negative := #NegEdge.Q;
	    
	END_REGION
	
END_FUNCTION_BLOCK
END_NAMESPACE

NAMESPACE Global
FUNCTION_BLOCK DataMan262
{ S7_Optimized_Access := 'TRUE' ; Published := 'TRUE' }
VERSION : 0.1
   VAR_INPUT 
      TriggerSignal : Bool;
      ContinuousGetResults : Bool;
      "Dataman-Results Available" : Bool;
      "Dataman-TriggerReady" : Bool;
      "Dataman-TriggerAck" : Bool;
      "Dataman-Train Focus Ack" : Bool;
      "Dataman-Train Match String Ack" : Bool;
      "Dataman-Execute DMCC Ack" : Bool;
      "Dataman-Set Match String Ack" : Bool;
      "Dataman-ResultID" : Int;
      "Dataman-Result Code" : Int;
      "Dataman-Result Length" : Int;
      "Result Data" : BarCode;
   END_VAR

   VAR_OUTPUT 
      "Dataman-UserData Length" : Word;
      "Dataman-UserData Option" : Word;
      "User Data" : BarCode;
   END_VAR

   VAR_IN_OUT 
      "Dataman-TriggerEnable" : Bool;
      "Dataman-Trigger" : Bool;
      "Dataman-ResultsAck" : Bool;
      "Dataman-Train Focus" : Bool;
      "Dataman-Train Match String" : Bool;
      "Dataman-Execute DMCC" : Bool;
      "Dataman-Set Match String" : Bool;
   END_VAR

   VAR 
      "Result Pending" : Bool;
      "Latest Results" : Struct
         ID : Int;
         Flags : Int;
         Length : Int;
         Value : Array[0..63] of Byte;
      END_STRUCT;
      "Train Focus" : Bool;
      "Train MatchString" : Bool;
      "Execute DMCC" : Bool;
      "Set Match String" : Bool;
      "String" : String[64] := '||>REBOOT$R$L';
      "Match String" : Array[0..63] of Byte;
      "Char" : Array[0..63] of Byte;
      Ret_val_1 { ExternalAccessible := 'False'; ExternalVisible := 'False'; ExternalWritable := 'False'} : Byte;
      R_TRIG_SimpleRead {InstructionName := 'R_TRIG'; LibVersion := '1.0'} : R_TRIG;
      R_TRIG_TrainFocus {InstructionName := 'R_TRIG'; LibVersion := '1.0'} : R_TRIG;
      "R_TRIG_Train MatchString" {InstructionName := 'R_TRIG'; LibVersion := '1.0'} : R_TRIG;
      R_TRIG_ExcuteDMCC {InstructionName := 'R_TRIG'; LibVersion := '1.0'} : R_TRIG;
      R_TRIG_SetMatchString {InstructionName := 'R_TRIG'; LibVersion := '1.0'} : R_TRIG;
      HoldTrigger { S7_SetPoint := 'True'} : Bool;
      HoldTrainFocus : Bool;
      HoldTrainMatchString : Bool;
      HoldDMCCExcute : Bool;
      HoldSetMatchString : Bool;
      ResultStr : String;
   END_VAR


BEGIN
	// ==========================================================================================================================================
	// Company        : LogTech, s.r.o.
	// Created by     : Mahmoud Elnady
	// Block          : FC_UpstreaProductionTote
	// Project        : Lekarna, Chrudim -PLC001 -MCC001
	// Project number : 23-157
	// ==========================================================================================================================================
	
	// This block will wait FOR the camera TO become ready, issue a trigger, wait FOR
	//the read TO complete AND THEN copy the read results TO DB5 ("LatestResults").
	//Trigger a read and retrieve the result data.
	REGION Simple Read
	           //Trigger a read and retrieve the result data.      
	    #R_TRIG_SimpleRead(CLK:=#TriggerSignal AND
	                       NOT #ContinuousGetResults);
	    IF #R_TRIG_SimpleRead.Q THEN
	        #HoldTrigger := TRUE;
	    END_IF;
	           
	    IF #HoldTrigger
	           THEN
	               //Make sure triggering is enabled 
	               REGION Triggering is Enabled 
	                   IF NOT #"Dataman-TriggerEnable" THEN
	                       #"Dataman-TriggerEnable" := TRUE;
	                   END_IF;
	               END_REGION
	               
	               //Special case (step 1): If results were already waiting before we issued a 
	               //trigger, process those results before starting a new read sequence.
	               REGION Process Results
	                   IF #"Dataman-Results Available" AND
	                       NOT #"Result Pending"
	                   THEN
	                       #"Result Pending" := TRUE;
	                       #"Dataman-ResultsAck" := TRUE;
	                   END_IF;
	                   
	               END_REGION
	               
	               //If camera ready and trigger not already issued, issue trigger signal. 
	               REGION Trigger Signal
	                   IF #"Dataman-TriggerReady" AND
	                       NOT #"Dataman-Trigger" AND
	                       NOT #"Dataman-TriggerAck" AND
	                       NOT #"Dataman-Results Available" AND
	                       NOT #"Dataman-ResultsAck" AND
	                       NOT #"Result Pending"
	                   THEN
	                       #"Dataman-Trigger" := TRUE;
	                       #"Result Pending" := TRUE;
	                   END_IF;
	                   
	               END_REGION
	               
	               //If results available, get the read results
	               REGION Read results
	                   IF #"Result Pending" AND
	                       #"Dataman-Results Available" AND
	                       NOT #"Dataman-ResultsAck"
	                   THEN
	                       #"Dataman-Trigger" := FALSE;
	                       #"Dataman-ResultsAck" := TRUE;
	                       #"Latest Results".ID := #"Dataman-ResultID";
	                       #"Latest Results".Flags := #"Dataman-Result Code";
	                       #"Latest Results".Length := #"Dataman-Result Length";
	                       MOVE_BLK(IN := #"Result Data"."Result Data"[0],
	                                COUNT := 64,
	                                OUT => #"Latest Results".Value[0]);
	                       
	                       //Convert last result data to value
	                       Chars_TO_Strg(Chars := #"Latest Results".Value,
	                                     pChars := 0,
	                                     Cnt := #"Latest Results".Length,
	                                     Strg => #ResultStr);
	                   END_IF;
	                   
	               END_REGION
	               
	               //Reset trigger signal as soon as it is acknowledged
	               //Reset results acknowledge signal as soon as it is recognized BY the reader.
	               
	               //This is the end OF the read sequence. Reset the "results pending" flag, set the
	               //output TO signal the operation is complete.
	               
	               //Note, the reader signals "results acknowledge" BY setting "results available" TO zero.
	               
	               REGION Reset trigger
	                   
	                   IF #"Result Pending" AND
	                           #"Dataman-ResultsAck" AND
	                           NOT #"Dataman-Results Available"
	                       THEN
	                           #"Dataman-ResultsAck" := FALSE;
	                           #"Result Pending" := FALSE;
	                           #HoldTrigger := FALSE;
	                       END_IF;
	                       
	               END_REGION
	               
	           END_IF;
	       END_REGION
	       
	//Read result data which was triggered elsewhere (i.e. manual trigger button)
	REGION Results Only
	           IF #ContinuousGetResults AND
	               NOT #TriggerSignal
	           THEN
	               
	               //IF results available, save the read results AND issue an acknowledge
	               REGION manual trigger button
	                   IF  #"Dataman-Results Available" AND
	                       NOT #"Dataman-ResultsAck"
	                   THEN
	                       #"Dataman-ResultsAck" := TRUE;
	                       #"Latest Results".ID := #"Dataman-ResultID";
	                       #"Latest Results".Flags := #"Dataman-Result Code";
	                       #"Latest Results".Length := #"Dataman-Result Length";
	                       MOVE_BLK(IN := #"Result Data"."Result Data"[0],
	                                COUNT := 64,
	                                OUT => #"Latest Results".Value[0]);
	                   END_IF;
	                   
	               END_REGION
	               
	               //IF the result acknowledge is complete, reset the result signal
	               REGION Reset signal
	                   IF #"Dataman-ResultsAck" AND
	                       NOT #"Dataman-Results Available"
	                   THEN
	                       #"Dataman-ResultsAck" := FALSE;
	                   END_IF;
	               END_REGION
	           END_IF;
	       END_REGION
	
	//Perform "Train Focus" operation.
	//Note, this operation only enables the training TO occur. After
	//executing this call the reader must be triggered TO perform the actual training.
	
	REGION Train Focus
	    //Perform "Train Focus" operation.
	    #R_TRIG_TrainFocus(CLK:=#"Train Focus");
	    
	    IF #R_TRIG_TrainFocus.Q THEN
	        #HoldTrainFocus := TRUE;
	    END_IF;
	    
	    IF #HoldTrainFocus THEN
	               REGION Initiate the "Train Focus"
	                   //Initiate the "Train Focus" operation AND monitor it TO completion.
	                   IF  NOT #"Dataman-Train Focus" AND
	                       NOT #"Dataman-Train Focus Ack"
	                   THEN
	                       #"Dataman-Train Focus" := True;
	                   END_IF;
	                   
	               END_REGION
	               
	               //Release "Train Focus" signal as soon as it is acknowledged by the reader
	               REGION Release "Train Focus"
	                   
	                   IF #"Dataman-Train Focus Ack" THEN
	                       #"Dataman-Train Focus" := FALSE;
	                       #HoldTrainFocus := FALSE;
	                   END_IF;
	                   
	               END_REGION
	           END_IF;
	       END_REGION
	
	
	//Perform "Train Match String" operation.
	//Note, this operation only enables the training TO occur. After
	//executing this call the reader must be triggered TO perform
	//the actual training.
	
	REGION Train MatchString
	    //Perform "Train Match String" operation.
	    #"R_TRIG_Train MatchString"(CLK:=#"Train MatchString");
	    
	    IF #"R_TRIG_Train MatchString".Q THEN
	        #HoldTrainMatchString := TRUE;
	    END_IF;
	    
	    IF  #HoldTrainMatchString THEN
	       //Issue "Train Match String" signal. 
	       REGION Issue Train Match String
	              IF  NOT #"Dataman-Train Match String" AND
	                       NOT #"Dataman-Train Match String Ack"
	                   THEN
	                       #"Dataman-Train Match String" := TRUE;
	              END_IF;
	       END_REGION
	               
	       //Release "Train Match String" signal as soon as it is acknowledged by the reader.
	       REGION Release "Train Match String"
	              IF #"Dataman-Train Match String Ack" THEN
	                  #"Dataman-Train Match String" := FALSE;
	                  #HoldTrainMatchString := FALSE;
	              END_IF;
	       END_REGION
	   END_IF;
	   
	END_REGION
	
	REGION DMCC Execute
	    //Perform "Execute DMCC" operation.
	    #R_TRIG_ExcuteDMCC(CLK := #"Execute DMCC");
	    
	    IF #R_TRIG_ExcuteDMCC.Q THEN
	        #HoldDMCCExcute := TRUE;
	    END_IF;
	    
	    IF #HoldDMCCExcute THEN
	        //Copy the DMCC command, and then issue the "DMCC Execute" signal.
	        REGION issue the "DMCC Execute"
	            
	            IF  NOT #"Dataman-Execute DMCC" AND
	                NOT #"Dataman-Execute DMCC Ack"
	            THEN
	                #"Dataman-Execute DMCC" := TRUE;
	                #"Dataman-UserData Length" := LEN(#String);
	                
	                Strg_TO_Chars(Strg := #String,
	                              pChars := 0,
	                              Cnt => #"Dataman-UserData Length",
	                              Chars := #"Match String");
	                
	                MOVE_BLK(IN := #"Match String"[0],
	                         COUNT := 64,
	                         OUT => #"User Data"."Result Data"[0]);
	            END_IF;
	            
	        END_REGION
	        
	        //Release "Execute DMCC" signal as soon as it is acknowledged by the reader.
	        REGION Release "Execute DMCC"
	            
	            IF #"Dataman-Execute DMCC Ack" THEN
	                #"Dataman-Execute DMCC" := FALSE;
	                #HoldDMCCExcute := FALSE;
	            END_IF;
	            
	        END_REGION
	    END_IF;
	END_REGION
	
	
	//Perform "Set Match String" operation.
	
	//Set the match String option, copy the Match String value, AND THEN issue "SetMatchString" signal.
	
	//Note, The symbology target's set are selected BY the value OF "UserDataOption".
	//0 = Set all symbologies
	//1 = Set only 2D
	//2 = Set only QR
	//3 = Set only 1D/stacked/postal
	
	REGION Set Match String
	    //Perform "Set Match String" operation.
	    #R_TRIG_SetMatchString(CLK:=#"Set Match String");
	    
	    IF #R_TRIG_SetMatchString.Q THEN
	        #HoldSetMatchString := TRUE;
	    END_IF;
	    
	    IF  #HoldSetMatchString THEN
	        REGION Set the match String option
	            IF NOT #"Dataman-Set Match String" AND
	                NOT #"Dataman-Set Match String Ack"
	            THEN
	                #"Dataman-Set Match String" := TRUE;
	                #"Dataman-UserData Option" := 1;
	                #"Dataman-UserData Length" := LEN(#String);
	                
	                Strg_TO_Chars(Strg := #String,
	                              pChars := 0,
	                              Cnt => #"Dataman-UserData Length",
	                              Chars := #Char);
	                
	                #Ret_val_1 := MOVE_BLK_VARIANT(SRC := #Char[0],
	                                               COUNT := 64,
	                                               SRC_INDEX := 0,
	                                               DEST_INDEX := 0,
	                                               DEST => #"Match String"[0]);
	                
	                MOVE_BLK(IN := #"Match String"[0],
	                         COUNT := 64,
	                         OUT => #"User Data"."Result Data"[0]);
	            END_IF;
	            
	        END_REGION
	        
	        //Release "SetMatchString" signal as soon as it is acknowledged BY the reader.
	        REGION Release "SetMatchString"
	            
	            IF #"Dataman-Set Match String Ack" THEN
	                #"Dataman-Set Match String" := FALSE;
	                #HoldSetMatchString := FALSE;
	            END_IF;
	            
	        END_REGION
	    END_IF;
	END_REGION
	
	
	
	
	
	
END_FUNCTION_BLOCK
END_NAMESPACE

NAMESPACE Global
FUNCTION_BLOCK FB_Klaxon
{ S7_Optimized_Access := 'TRUE' ; Published := 'TRUE' }
VERSION : 0.1
   VAR_INPUT 
      SystemStart : Bool;
      SystemStop : Bool;
      ReadGlobalFault : Bool;
      ReadGlobalReady : Bool;
      ReadEstopActive : Bool;
      ReadGlobalBlockage : Bool;
   END_VAR

   VAR 
      KLAXON_HORN : FB_KlaxonHorn;
      KLAXON_YELLOW : FB_KlaxonLampYellow;
      HORN : Bool;
      YELLOW : Bool;
      GREEN : Bool;
   END_VAR


BEGIN
	// ==========================================================================================================================================================================
	// Company       : LogTech, s.r.o.
	// Created by    : Anton Vinoth Soundraraj
	// Block         : FB_Klaxon
	// Project       : LT-LIB-Block
	// ==========================================================================================================================================================================
	
	REGION Klaxon Horn
	    
	    // FB_KlaxonHorn
	    // Called as MIDB
	    
	    #KLAXON_HORN(Start          := #SystemStart,
	                 Stop           := #SystemStop,
	                 GlobalFault    := #ReadGlobalFault,
	                 GlobalBlockage := #ReadGlobalBlockage,
	                 EstopActive    := #ReadEstopActive,
	                 HornActive     => #HORN);
	    
	END_REGION
	
	REGION Klaxon Yellow
	    
	    // FB_KlaxonLampYellow
	    // Called as MIDB
	    
	    #KLAXON_YELLOW(BlinkCondition := #SystemStart,
	                   GlowCondition  := NOT #ReadGlobalReady,
	                   BlockageStatus := #ReadGlobalBlockage,
	                   YellowLamp     => #YELLOW);
	    
	END_REGION
	
	REGION Klaxon Green
	    
	    #GREEN :=
	    #ReadGlobalReady AND
	    NOT #ReadGlobalBlockage AND
	    NOT #KLAXON_YELLOW.StartupActive AND 
	    NOT #KLAXON_YELLOW.YellowLamp;
	    
	END_REGION
END_FUNCTION_BLOCK
END_NAMESPACE

NAMESPACE Global
FUNCTION_BLOCK FB_KlaxonHorn
{ S7_Optimized_Access := 'TRUE' ; Published := 'TRUE' }
VERSION : 0.1
   VAR_INPUT 
      Start : Bool;
      Stop : Bool;
      GlobalFault : Bool;
      GlobalBlockage : Bool;
      EstopActive : Bool;
      Fire : Bool;
   END_VAR

   VAR_OUTPUT 
      HornActive : Bool;
   END_VAR

   VAR 
      RT_Start {InstructionName := 'R_TRIG'; LibVersion := '1.0'; S7_SetPoint := 'False'} : R_TRIG;
      RT_Stop {InstructionName := 'R_TRIG'; LibVersion := '1.0'} : R_TRIG;
      RT_Estop {InstructionName := 'R_TRIG'; LibVersion := '1.0'} : R_TRIG;
      RT_Fault {InstructionName := 'R_TRIG'; LibVersion := '1.0'} : R_TRIG;
      RT_Blockage {InstructionName := 'R_TRIG'; LibVersion := '1.0'} : R_TRIG;
      RT_Fire {InstructionName := 'R_TRIG'; LibVersion := '1.0'} : R_TRIG;
      KlaxonHornTimer {InstructionName := 'IEC_TIMER'; LibVersion := '1.0'; S7_SetPoint := 'False'} : IEC_TIMER;
      KlaxonHornCondition { S7_SetPoint := 'True'} : Bool;
      HornCondition : Bool;
   END_VAR


BEGIN
	// ==========================================================================================================================================================================
	// Company      : LogTech, s.r.o.
	// Created by   : Anton Vinoth Soundraraj
	// Project      : LT-Lib-Block
	// Block        : FB_KlaxonHorn
	// ==========================================================================================================================================================================
	
	REGION Horn
	    
	    // trigger kaxon horn: rising trigger of start
	    #RT_Start(CLK := #Start);
	    // trigger kaxon horn: rising trigger of stop
	    #RT_Stop(CLK := #Stop);
	    // trigger kaxon horn: rising trigger of fault
	    #RT_Fault(CLK := #GlobalFault);
	    // trigger kaxon horn: rising trigger of blockage
	    #RT_Blockage(CLK := #GlobalBlockage);
	    // trigger kaxon horn: rising trigger of estop
	    #RT_Estop(CLK := #EstopActive);
	    // trigger kaxon horn: rising trigger of fire
	    #RT_Fire(CLK := #Fire);
	    
	    // --------------
	    // Horn condition
	    // --------------
	    
	    #HornCondition :=
	    #RT_Start.Q OR
	    #RT_Stop.Q OR
	    #RT_Fire.Q OR
	    #RT_Fault.Q OR
	    #RT_Estop.Q OR
	    #RT_Fire.Q;
	    
	    // -------------------
	    // Horn alert duration
	    // -------------------
	    
	    #KlaxonHornTimer.TOF(IN := #HornCondition,
	                         PT := t#5s);
	    
	    #HornActive :=
	    #KlaxonHornTimer.Q;
	    
	END_REGION
	
	
	
	
	
	
	
	
	
	
	
	
	
END_FUNCTION_BLOCK
END_NAMESPACE

NAMESPACE ProductionLine
FUNCTION_BLOCK Flow_Test
{ S7_Optimized_Access := 'TRUE' ; Published := 'FALSE' }
VERSION : 0.1
   VAR 
      Start { S7_SetPoint := 'True'} : Bool;   //  // Start command (e.g. from I0.0)
      StartTest : Test_Logic;
      GoToRightDP1 : Test_Logic;
      ContinueStraightDP1 : Test_Logic;
      ContinueStraightDP2 : Test_Logic;
      GotorightDP2Thentoright : Test_Logic;
      GotorightDP2ThentoLeft : Test_Logic;
      ContinueStraightDP3 : Test_Logic;
      ContinueStraightDP4 : Test_Logic;
      GotoRightDP4 : Test_Logic;
      "A1.13.1_Straight" : Test_Logic;
      "A1.13.1_left" : Test_Logic;
      R_TRIG_Instance {InstructionName := 'R_TRIG'; LibVersion := '1.0'} : R_TRIG;
   END_VAR


BEGIN
	// ==========================================================================================================================================
	// Company        : LogTech, s.r.o.
	// Created by     : Mahmoud Elnady
	// Block          : FB_FlowTest
	// Project        : Lékárna Chrudim
	// Project number : 23-157
	// ==========================================================================================================================================
	
	REGION Start Test
	    #StartTest(Start := #Start,
	               StartPoint := _."A1.1.1",
	               EndPoint :=  _."A1.5.3");
	END_REGION
	
	
	REGION Go TO Right DP1
	    #GoToRightDP1(Start := DB_ToteTracking.Conveyor[_."A1.6.1"].ToteDir.toRight AND
	                  DB_ToteTracking.Conveyor[_."A1.6.2"].ToteDir.toRight AND
	                  _.ProductionLine.IDB_ProductionLine."A1.5.3".FilteredSensor,
	                  StartPoint := _."B1.1.1",
	                  EndPoint := _."B1.9.2");
	END_REGION
	
	
	REGION CONTINUE Straight DP1
	    
	    #ContinueStraightDP1(Start := DB_ToteTracking.Conveyor[_."A1.6.1"].ToteDir.Straight AND
	                         DB_ToteTracking.Conveyor[_."A1.6.2"].ToteDir.Straight AND
	                         _.ProductionLine.IDB_ProductionLine."A1.5.3".FilteredSensor,
	                         StartPoint := _."A1.7.1",
	                         EndPoint := _."A1.8.1");
	    
	END_REGION
	
	IF (DB_ToteTracking.Conveyor[_."A1.6.1"].ToteDir.Straight OR
	    DB_ToteTracking.Conveyor[_."A1.6.1"].ToteDir.toRight) AND
	    IDB_ProductionLine."A1.5.3".FilteredSensor
	THEN
	    _.Global.DB_SystemSimu.TriggerSensor.Line.ProductionLine.Conveyor[_."A1.6.1"] := TRUE;
	ELSE
	    _.Global.DB_SystemSimu.TriggerSensor.Line.ProductionLine.Conveyor[_."A1.6.1"] := FALSE;
	END_IF;
	
	
	        
	REGION CONTINUE Straight DP2
	    
	    #ContinueStraightDP2(Start := DB_ToteTracking.Conveyor[_."B1.10.1"].ToteDir.Straight AND
	                                  IDB_ProductionLine."B1.9.2".FilteredSensor,
	                         StartPoint := _."B1.11.1",
	                         EndPoint := _."B1.17.4");
	    
	END_REGION
	
	
	REGION Go TO Right DP2 THEN TO Right
	    #GotorightDP2Thentoright(Start := DB_ToteTracking.Conveyor[_."B1.10.1"].ToteDir.toRight AND
	                             DB_ToteTracking.Conveyor[_."C1.3.1"].ToteDir.toRight AND
	                             IDB_ProductionLine."B1.9.2".FilteredSensor,
	                             StartPoint := _."C1.2.2",
	                             EndPoint := _."C1.2.1");
	END_REGION
	
	
	REGION Go TO Right THEN TO Left
	    #GotorightDP2ThentoLeft(Start := DB_ToteTracking.Conveyor[_."B1.10.1"].ToteDir.toRight AND
	                            DB_ToteTracking.Conveyor[_."C1.3.1"].ToteDir.toLeft AND
	                            IDB_ProductionLine."B1.9.2".FilteredSensor,
	                            StartPoint := _."C1.4.1",
	                            EndPoint :=  _."C1.4.2");
	END_REGION
	
	
	IF (DB_ToteTracking.Conveyor[_."B1.10.1"].ToteDir.Straight OR
	    DB_ToteTracking.Conveyor[_."B1.10.1"].ToteDir.toRight) AND
	    IDB_ProductionLine."B1.9.2".FilteredSensor
	THEN
	    _.Global.DB_SystemSimu.TriggerSensor.Line.ProductionLine.Conveyor[_."B1.10.1"] := TRUE;
	ELSE
	    _.Global.DB_SystemSimu.TriggerSensor.Line.ProductionLine.Conveyor[_."B1.10.1"] := FALSE;
	END_IF;
	
	IF (DB_ToteTracking.Conveyor[_."C1.3.1"].ToteDir.toLeft OR
	    DB_ToteTracking.Conveyor[_."C1.3.1"].ToteDir.toRight) AND
	    IDB_ProductionLine."B1.10.1".FilteredSensor AND
	    DB_ToteTracking.Conveyor[_."B1.10.1"].ToteDir.toRight
	THEN
	    _.Global.DB_SystemSimu.TriggerSensor.Line.ProductionLine.Conveyor[_."C1.3.1"] := TRUE;
	ELSE
	    _.Global.DB_SystemSimu.TriggerSensor.Line.ProductionLine.Conveyor[_."C1.3.1"] := FALSE;
	END_IF;
	
	
	
	REGION CONTINUE Straight DP3
	    #ContinueStraightDP3(Start := DB_ToteTracking.Conveyor[_."B1.18.1"].ToteDir.Straight AND
	                                  IDB_ProductionLine."B1.17.4".FilteredSensor,
	                         StartPoint := _."B1.19.1",
	                         EndPoint := _."B1.23.1");
	END_REGION
	
	IF (DB_ToteTracking.Conveyor[_."B1.18.1"].ToteDir.toLeft OR
	    DB_ToteTracking.Conveyor[_."B1.18.1"].ToteDir.Straight) AND
	    IDB_ProductionLine."B1.17.4".FilteredSensor
	THEN
	    _.Global.DB_SystemSimu.TriggerSensor.Line.ProductionLine.Conveyor[_."B1.18.1"] := TRUE;
	ELSE
	    _.Global.DB_SystemSimu.TriggerSensor.Line.ProductionLine.Conveyor[_."B1.18.1"] := FALSE;
	END_IF;
	
	#R_TRIG_Instance(CLK:=( IDB_ProductionLine."B1.18.1".FilteredSensor AND
	                 DB_ToteTracking.Conveyor[_."B1.18.1"].ToteDir.toLeft));
	
	
	
	REGION CONTINUE Straight DP4
	    #ContinueStraightDP4(Start := DB_ToteTracking.Conveyor[_."A1.9.1"].ToteDir.Straight AND
	                         DB_ToteTracking.Conveyor[_."A1.9.2"].ToteDir.Straight AND
	                         _.ProductionLine.IDB_ProductionLine."A1.8.1".FilteredSensor,
	                         StartPoint := _."A1.10.1",
	                         EndPoint := _."A1.12.2");
	END_REGION
	
	
	REGION Go TO Right DP4
	    #GotoRightDP4(Start := DB_ToteTracking.Conveyor[_."A1.9.1"].ToteDir.toRight AND
	                  DB_ToteTracking.Conveyor[_."A1.9.2"].ToteDir.toRight AND
	                  _.ProductionLine.IDB_ProductionLine."A1.8.1".FilteredSensor,
	                  StartPoint := _."D1.1.1",
	                  EndPoint :=  _."D1.12.3");
	END_REGION
	
	IF (DB_ToteTracking.Conveyor[_."A1.9.1"].ToteDir.Straight OR
	    DB_ToteTracking.Conveyor[_."A1.9.1"].ToteDir.toRight) AND
	    IDB_ProductionLine."A1.8.1".FilteredSensor
	THEN
	    _.Global.DB_SystemSimu.TriggerSensor.Line.ProductionLine.Conveyor[_."A1.9.1"] := TRUE;
	ELSE
	    _.Global.DB_SystemSimu.TriggerSensor.Line.ProductionLine.Conveyor[_."A1.9.1"] := FALSE;
	END_IF;
	
	REGION A1.13.1_Straight
	    
	    #"A1.13.1_Straight"(Start:= DB_ToteTracking.Conveyor[_."A1.13.1"].ToteDir.Straight AND
	                                IDB_ProductionLine."A1.12.2".FilteredSensor,
	                        StartPoint:=_."A1.14.1",
	                        EndPoint:= _."A1.14.26");
	    
	   
	END_REGION
	        
	REGION A1.13.1_Left
	    
	    #"A1.13.1_left"(Start := DB_ToteTracking.Conveyor[_."A1.13.1"].ToteDir.toLeft AND
	                    IDB_ProductionLine."A1.12.2".FilteredSensor,
	                    StartPoint := _."A2.2.1",
	                    EndPoint := _."A2.2.26");
	    
	    
	END_REGION
	
	
	    
	    
	
END_FUNCTION_BLOCK
END_NAMESPACE

NAMESPACE ProductionLine
FUNCTION_BLOCK Test_Logic
{ S7_Optimized_Access := 'TRUE' ; Published := 'FALSE' }
VERSION : 0.1
   VAR_INPUT 
      Start : Bool;
      StartPoint : Int;
      EndPoint : Int;
   END_VAR

   VAR 
      Active : Bool;
      "Counter" : Int;
      PulseTimer {InstructionName := 'TON_TIME'; LibVersion := '1.0'; S7_SetPoint := 'False'} : TON_TIME;
   END_VAR


BEGIN
	// ==========================================================================================================================================
	// Company        : LogTech, s.r.o.
	// Created by     : Mahmoud Elnady
	// Block          : FB_LineA1
	// Project        : Lékárna Chrudim
	// Project number : 23-157
	// ==========================================================================================================================================
	
	REGION Start
	    // Start sequence
	    IF #Start AND NOT #Active THEN
	        #Active := TRUE;
	        #Counter := #StartPoint;               // Start from first output
	    END_IF;
	    
	    // Main pulse logic
	    IF #Active THEN
	        // Turn ON the current output
	        _.Global.DB_SystemSimu.TriggerSensor.Line.ProductionLine.Conveyor[#Counter] := TRUE;
	        #PulseTimer(IN := TRUE,
	                    PT := T#3s);
	        
	        // When timer expires
	        IF #PulseTimer.Q THEN
	            // Turn OFF current output
	            _.Global.DB_SystemSimu.TriggerSensor.Line.ProductionLine.Conveyor[#Counter] := FALSE;
	            
	            // Reset timer
	            RESET_TIMER(#PulseTimer);
	            
	            // Move to next output
	            #Counter := #Counter + 1;
	            
	            // Stop if last output finished
	            IF #Counter > #EndPoint THEN
	                #Active := FALSE;
	            END_IF;
	        END_IF;
	    ELSE
	        // Make sure all outputs are OFF when not active
	        (* FOR #var_i := 1001 TO #N DO
	        //#Q[#var_i] := FALSE;
	        _.Global.DB_SystemSimu.TriggerSensor.Line.ProductionLine.Conveyor[#Counter] := FALSE;
	    END_FOR;*)
	        RESET_TIMER(#PulseTimer);
	    END_IF;
	END_REGION
END_FUNCTION_BLOCK
END_NAMESPACE

NAMESPACE ProductionLine
FUNCTION_BLOCK BarcodeReader
{ S7_Optimized_Access := 'TRUE' ; Published := 'FALSE' }
VERSION : 0.1
   VAR 
      DP1 { S7_SetPoint := 'False'} : _.Global.DataMan262;
      DP2 { S7_SetPoint := 'False'} : _.Global.DataMan262;
      DP3 { S7_SetPoint := 'False'} : _.Global.DataMan262;
      DP4 { S7_SetPoint := 'False'} : _.Global.DataMan262;
   END_VAR


BEGIN
	// ==========================================================================================================================================
	// Company        : LogTech, s.r.o.
	// Created by     : Mahmoud Elnady
	// Block          : Barcode Reader
	// Project        : Lekarna, Chrudim -PLC001 -MCC001
	// Project number : 23-157
	// ==========================================================================================================================================
	
	REGION DP1
	    
	    #DP1(TriggerSignal:= IDB_ProductionLine."A1.5.1".FilteredSensor,
	         "Dataman-Results Available":=_."DP1-Results Available",
	         "Dataman-TriggerReady":=_."DP1-TriggerReady",
	         "Dataman-TriggerAck":=_."DP1-TriggerAck",
	         "Dataman-ResultID":=_."DP1-ResultID",
	         "Dataman-Result Code":=_."DP1-Result Code",
	         "Dataman-Result Length":=_."DP1-Result Length",
	         "Result Data":=_."Result data_DP1",
	         "Dataman-UserData Length"=>_."DP1-UserData Length",
	         "Dataman-UserData Option"=>_."DP1-UserData Option",
	         "User Data"=>_.UserData_DP1,
	         "Dataman-TriggerEnable":=_."DP1-TriggerEnable",
	         "Dataman-Trigger":=_."DP1-Trigger",
	         "Dataman-ResultsAck":=_."DP1-ResultsAck");
	    
	END_REGION
	
	REGION DP2
	    
	    #DP2(TriggerSignal := IDB_ProductionLine."B1.9.1".FilteredSensor,
	         "Dataman-Results Available" := _."DP2-Results Available",
	         "Dataman-TriggerReady" := _."DP2-TriggerReady",
	         "Dataman-TriggerAck" := _."DP2-TriggerAck",
	         "Dataman-ResultID" := _."DP2-ResultID",
	         "Dataman-Result Code" := _."DP2-Result Code",
	         "Dataman-Result Length" := _."DP2-Result Length",
	         "Result Data" := _."Result data_DP2",
	         "Dataman-UserData Length" => _."DP2-UserData Length",
	         "Dataman-UserData Option" => _."DP2-UserData Option",
	         "User Data" => _.UserData_DP2,
	         "Dataman-TriggerEnable" := _."DP2-TriggerEnable",
	         "Dataman-Trigger" := _."DP2-Trigger",
	         "Dataman-ResultsAck" := _."DP2-ResultsAck");
	    
	END_REGION
	
	REGION DP3
	    
	    #DP3(TriggerSignal := IDB_ProductionLine."B1.17.1".FilteredSensor,
	         "Dataman-Results Available" := _."DP3-Results Available",
	         "Dataman-TriggerReady" := _."DP3-TriggerReady",
	         "Dataman-TriggerAck" := _."DP3-TriggerAck",
	         "Dataman-ResultID" := _."DP3-ResultID",
	         "Dataman-Result Code" := _."DP3-Result Code",
	         "Dataman-Result Length" := _."DP3-Result Length",
	         "Result Data" := _."Result data_DP3",
	         "Dataman-UserData Length" => _."DP3-UserData Length",
	         "Dataman-UserData Option" => _."DP3-UserData Option",
	         "User Data" => _.UserData_DP3,
	         "Dataman-TriggerEnable" := _."DP3-TriggerEnable",
	         "Dataman-Trigger" := _."DP3-Trigger",
	         "Dataman-ResultsAck" := _."DP3-ResultsAck");
	    
	END_REGION
	
	
	REGION DP4
	    
	    #DP4(TriggerSignal := IDB_ProductionLine."A1.7.4".FilteredSensor,
	         "Dataman-Results Available" := _."DP4-Results Available",
	         "Dataman-TriggerReady" := _."DP4-TriggerReady",
	         "Dataman-TriggerAck" := _."DP4-TriggerAck",
	         "Dataman-ResultID" := _."DP4-ResultID",
	         "Dataman-Result Code" := _."DP4-Result Code",
	         "Dataman-Result Length" := _."DP4-Result Length",
	         "Result Data" := _."Result data_DP4",
	         "Dataman-UserData Length" => _."DP4-UserData Length",
	         "Dataman-UserData Option" => _."DP4-UserData Option",
	         "User Data" => _.UserData_DP4,
	         "Dataman-TriggerEnable" := _."DP4-TriggerEnable",
	         "Dataman-Trigger" := _."DP4-Trigger",
	         "Dataman-ResultsAck" := _."DP4-ResultsAck");
	    
	END_REGION
	
END_FUNCTION_BLOCK
END_NAMESPACE

NAMESPACE ProductionLine
FUNCTION_BLOCK FB_OPC_Communication
{ S7_Optimized_Access := 'TRUE' ; Published := 'FALSE' }
VERSION : 0.1
   VAR 
      Communication_DP1 { S7_SetPoint := 'False'} : FB_OPC_DestRequest;
      Communication_DP2 { S7_SetPoint := 'False'} : FB_OPC_DestRequest;
      Communication_DP3 { S7_SetPoint := 'False'} : FB_OPC_DestRequest;
      Communication_DP4 { S7_SetPoint := 'False'} : FB_OPC_DestRequest;
      Communication_IP1 { S7_SetPoint := 'False'} : FB_OPC_DestInfo;
      Communication_IP2 { S7_SetPoint := 'False'} : FB_OPC_DestInfo;
      Communication_IP3 { S7_SetPoint := 'False'} : FB_OPC_DestInfo;
      Communication_IP4 { S7_SetPoint := 'False'} : FB_OPC_DestInfo;
      Communication_IP5 { S7_SetPoint := 'False'} : FB_OPC_DestInfo;
      Communication_IP6 { S7_SetPoint := 'False'} : FB_OPC_DestInfo;
      Communication_IP7 { S7_SetPoint := 'False'} : FB_OPC_DestInfo;
      Communication_IP8 { S7_SetPoint := 'False'} : FB_OPC_DestInfo;
      Communication_IP9 { S7_SetPoint := 'False'} : FB_OPC_DestInfo;
      Communication_SYS_OP { S7_SetPoint := 'False'} : FB_OPC_SysStatus;
      Communication_SYS_OP_Source : OPC_SystemStatus;
      Communication_SYS_OP_Ack : OPC_SystStatus_Ack;
      timPeriodicSend {InstructionName := 'IEC_TIMER'; LibVersion := '1.0'} : IEC_TIMER;
      timWatchdog {InstructionName := 'IEC_TIMER'; LibVersion := '1.0'} : IEC_TIMER;
      Communication_fault : Bool;
   END_VAR


BEGIN
	// ==========================================================================================================================================
	// Company        : LogTech, s.r.o.
	// Created by     : Mahmoud Elnady
	// Block          : FB_OPC_Communication
	// Project        : Lekarna, Chrudim -PLC001 -MCC001
	// Project number : 23-157
	// ==========================================================================================================================================
	
	//------------------------------------------------------
	// Initialization
	//------------------------------------------------------
	
	REGION Initialization
	    // Initialization section to reset the sequence numbers at the first scan
	    IF _.DB_Sync.memoryBit.FirstScan THEN
	        OPC_Data.DP1.DestRequest.Source.SourceSeq := 0;
	        OPC_Data.DP2.DestRequest.Source.SourceSeq := 0;
	        OPC_Data.DP3.DestRequest.Source.SourceSeq := 0;
	        OPC_Data.DP4.DestRequest.Source.SourceSeq := 0;
	        OPC_Data.IP1.DestInfo.Source.SourceSeq := 0;
	        OPC_Data.IP2.DestInfo.Source.SourceSeq := 0;
	        OPC_Data.IP3.DestInfo.Source.SourceSeq := 0;
	        OPC_Data.IP4.DestInfo.Source.SourceSeq := 0;
	        OPC_Data.IP5.DestInfo.Source.SourceSeq := 0;
	        OPC_Data.IP6.DestInfo.Source.SourceSeq := 0;
	        OPC_Data.IP7.DestInfo.Source.SourceSeq := 0;
	        OPC_Data.IP8.DestInfo.Source.SourceSeq := 0;
	        OPC_Data.IP9.DestInfo.Source.SourceSeq := 0;
	    END_IF;
	END_REGION
	
	//------------------------------------------------------
	// Handle destination request/ destination Information communication
	//------------------------------------------------------
	
	REGION DP1- DestRequest
	    // Handle destination request communication for DP1
	    #Communication_DP1(Source := OPC_Data.DP1.DestRequest.Source,
	                       Ack := OPC_Data.DP1.DestRequest.Ack);
	    
	END_REGION
	
	
	REGION DP2- DestRequest
	    // Handle destination request communication for DP2
	    #Communication_DP2(Source := OPC_Data.DP2.DestRequest.Source,
	                       Ack := OPC_Data.DP2.DestRequest.Ack);
	END_REGION
	
	
	REGION DP3- DestRequest
	    // Handle destination request communication for DP3
	    #Communication_DP3(Source := OPC_Data.DP3.DestRequest.Source,
	                       Ack := OPC_Data.DP3.DestRequest.Ack);
	END_REGION
	
	
	REGION DP4- DestRequest
	    // Handle destination request communication for DP4
	    #Communication_DP4(Source := OPC_Data.DP4.DestRequest.Source,
	                       Ack := OPC_Data.DP4.DestRequest.Ack);
	END_REGION
	
	REGION DS1- DestRequest
	    // Handle destination information communication for DS1
	    #Communication_IP1(Source := OPC_Data.IP1.DestInfo.Source,
	                       Ack := OPC_Data.IP1.DestInfo.Ack);
	END_REGION
	
	
	REGION DS2- DestRequest
	    // Handle destination information communication for DS2
	    #Communication_IP2(Source := OPC_Data.IP2.DestInfo.Source,
	                       Ack := OPC_Data.IP2.DestInfo.Ack);
	END_REGION
	
	
	REGION DS3- DestRequest
	    // Handle destination information communication for DS3
	    #Communication_IP3(Source := OPC_Data.IP3.DestInfo.Source,
	                       Ack := OPC_Data.IP3.DestInfo.Ack);
	END_REGION
	
	
	REGION DS4- DestRequest
	    // Handle destination information communication for DS4
	    #Communication_IP4(Source := OPC_Data.IP4.DestInfo.Source,
	                       Ack := OPC_Data.IP4.DestInfo.Ack);
	END_REGION
	
	REGION DS5- DestRequest
	    // Handle destination information communication for DS4
	    #Communication_IP5(Source := OPC_Data.IP5.DestInfo.Source,
	                       Ack := OPC_Data.IP5.DestInfo.Ack);
	END_REGION
	
	REGION DS6- DestRequest
	    // Handle destination information communication for DS4
	    #Communication_IP6(Source := OPC_Data.IP6.DestInfo.Source,
	                       Ack := OPC_Data.IP6.DestInfo.Ack);
	END_REGION
	
	REGION DS7- DestRequest
	    // Handle destination information communication for DS4
	    #Communication_IP7(Source := OPC_Data.IP7.DestInfo.Source,
	                       Ack := OPC_Data.IP7.DestInfo.Ack);
	END_REGION
	
	REGION DS8- DestRequest
	    // Handle destination information communication for DS4
	    #Communication_IP8(Source := OPC_Data.IP8.DestInfo.Source,
	                       Ack := OPC_Data.IP8.DestInfo.Ack);
	END_REGION
	
	REGION DS9- DestRequest
	    // Handle destination information communication for DS4
	    #Communication_IP9(Source := OPC_Data.IP9.DestInfo.Source,
	                       Ack := OPC_Data.IP9.DestInfo.Ack);
	END_REGION
	
	//------------------------------------------------------
	//Handle communication for overall system operation status
	//------------------------------------------------------
	
	REGION  SystStatus
	    // Statement section REGION
	    #Communication_SYS_OP(Source:=#Communication_SYS_OP_Source,
	                          Ack:=#Communication_SYS_OP_Ack);
	    
	END_REGION
	
	
	//------------------------------------------------------
	// Heart Beats
	//------------------------------------------------------
	
	REGION SYS Position - SystStatus
	    // // Periodic communication trigger for system status data (SYS_OP)
	    IF NOT #timPeriodicSend.Q THEN
	        #Communication_SYS_OP.Comm.Send := TRUE;
	    END_IF;
	    
	    #timPeriodicSend.TON(IN := #Communication_SYS_OP.Comm.Send AND
	                               #Communication_SYS_OP.Comm.Send_prev,
	                         PT := T#10s);
	    IF #timPeriodicSend.Q THEN
	        #Communication_SYS_OP.Comm.Send := FALSE;
	    END_IF;
	
	END_REGION
	
	//Periodic Counter, incremented every 10 seconds.
	//IF one side does NOT increment the counter within 30 seconds,
	//it will be considered offline BY the other side.
	REGION Watchdog
	    
	    OPC_Data.Watchdog.Keep_Alive_PLC := #Communication_SYS_OP.Comm.SourceSeq;
	    
	    #Communication_SYS_OP.Comm.AckSeq := OPC_Data.Watchdog.Keep_Alive_WMS;
	    
	END_REGION
	
	
	REGION Communication Fault
	    
	    #timWatchdog.TON(IN :=  #Communication_SYS_OP.Comm.SourceSeq <> #Communication_SYS_OP.Comm.AckSeq ,
	                          PT := T#30s);
	    
	    IF #timWatchdog.Q THEN
	        #Communication_fault := TRUE;
	    ELSE
	        #Communication_fault := FALSE;
	    END_IF;
	    
	END_REGION
	
	//------------------------------------------------------
	// Status of Segment for WMS
	//------------------------------------------------------
	
	REGION Status OF Segment FOR WMS
	    // Status of Segment for WMS
	    //Update system status based on Flow Rack Loop status
	    IF IDB_Segments_Status.FlowRackLoopReadyToRun THEN
	        // If conveyor is ready, set OPC system status to '1'
	        OPC_Data.Status.Segment.FlowRackLoop := 1;
	    ELSE
	        // If not ready, set system status to '0'
	        OPC_Data.Status.Segment.FlowRackLoop := 0;
	    END_IF;
	    
	    IF IDB_Segments_Status.FlowRackWorkPlaceRightReadyToRun THEN
	        OPC_Data.Status.Segment.FlowRackWorkplaceRight := 1;
	    ELSE
	        OPC_Data.Status.Segment.FlowRackWorkplaceRight := 0;
	    END_IF;
	    
	    IF IDB_Segments_Status.FlowRackWorkPlaceLeftReadyToRun THEN
	        OPC_Data.Status.Segment.FlowRackWorkplaceLeft := 1;
	    ELSE
	        OPC_Data.Status.Segment.FlowRackWorkplaceLeft := 0;
	    END_IF;
	    
	    IF IDB_Segments_Status.FragileloopReadyToRun THEN
	        OPC_Data.Status.Segment.FragileLoop := 1;
	    ELSE
	        OPC_Data.Status.Segment.FragileLoop := 0;
	    END_IF;
	    
	END_REGION
	
	
	
	
	
	
	
	
	
	
	
	
END_FUNCTION_BLOCK
END_NAMESPACE

NAMESPACE ProductionLine
FUNCTION_BLOCK FB_OPC_DestAssigne
{ S7_Optimized_Access := 'TRUE' ; Published := 'FALSE' }
VERSION : 0.1
   VAR_IN_OUT 
      Source : OPC_DestAssign;
      Ack : OPC_DestAssign_Ack;
   END_VAR

   VAR 
      Communication { S7_SetPoint := 'False'} : FB_OPC_ReceiveSendAck;
      staSource : OPC_DestAssign;
      staAck : OPC_DestAssign_Ack;
   END_VAR

   VAR_TEMP 
      Retval : Int;
   END_VAR


BEGIN
	// ==========================================================================================================================================
	// Company        : LogTech, s.r.o.
	// Created by     : Mahmoud Elnady
	// Block          : OPC_SendReciveAck
	// Project        : Lekarna, Chrudim -PLC001 -MCC001
	// Project number : 23-157
	// ==========================================================================================================================================
	
	//======================================================
	// Region: Communication Handling and Logging
	// Description: Manages the communication routine and logs
	//              events for message sending, acknowledgment
	//              reception, and acknowledgment timeout.
	//======================================================
	
	//------------------------------------------------------
	// Call communication routine
	//------------------------------------------------------
	
	REGION Communication routine
	    // Call communication routine
	    #Communication(SourceSeq := #staSource.SourceSeq,
	                   AckSeq := #staAck.AckSeq);
	END_REGION
	
	#Source.SourceSeq := #staSource.SourceSeq;
	#staAck.AckSeq := #Ack.AckSeq;
	
	
	//------------------------------------------------------
	// Log event when a new message is sent
	//------------------------------------------------------
	
	REGION Log event - new message
	    IF #Communication.Log.New_data_received THEN
	        #Communication.Log.New_data_received := FALSE;
	        // Logging
	        //(LOG)3005=$ Node $, new message received, seq: $, palletID: $, WMSID $, destination: $, no-stretch: $
	        DB_LogMsg.LogMsg_9.Para_STRING_01.Data := #Source.SourceNode;
	        DB_LogMsg.LogMsg_9.Para_BYTE_02.Data := #Source.SourceSeq;
	        DB_LogMsg.LogMsg_9.Para_STRING_03.Data := #Source.TotesID;
	        DB_LogMsg.LogMsg_9.Para_STRING_04.Data := #Source.WMSID;
	        DB_LogMsg.LogMsg_9.Para_STRING_05.Data := #Source.DestinationNode;
	        #Retval := FC_LogMsg(EventID := 3005, EventLevel := 2, EventGroup := 33, LogMsg := DB_LogMsg.LogMsg_9);
	    END_IF;
	END_REGION
	
	//------------------------------------------------------
	// Log event when new acknowledgment is received
	//------------------------------------------------------
	
	REGION Log event-New acknowledgment
	    IF #Communication.Log.Ack_send THEN
	        #Communication.Log.Ack_send := FALSE;
	        // Logging
	        //(LOG)3006=$ Node $, acknowledge sent, seq: $, palletID: $, WMSID: $, confirmation: $
	        DB_LogMsg.LogMsg_10.Para_STRING_01.Data := #Ack.SourceNode;
	        DB_LogMsg.LogMsg_10.Para_BYTE_02.Data := #Ack.AckSeq;
	        DB_LogMsg.LogMsg_10.Para_STRING_03.Data := #Ack.TotesID;
	        DB_LogMsg.LogMsg_10.Para_STRING_04.Data := #Ack.WMSID;
	        DB_LogMsg.LogMsg_10.Para_CHAR_05.Data := STRING_TO_CHAR(#Ack.Confirmation);
	        #Retval := FC_LogMsg(EventID := 3006, EventLevel := 2, EventGroup := 33, LogMsg := DB_LogMsg.LogMsg_10);
	    END_IF;
	END_REGION
	
	
END_FUNCTION_BLOCK
END_NAMESPACE

NAMESPACE ProductionLine
FUNCTION_BLOCK FB_OPC_DestInfo
{ S7_Optimized_Access := 'TRUE' ; Published := 'FALSE' }
VERSION : 0.1
   VAR_IN_OUT 
      Source : OPC_DestInfo;
      Ack : OPC_DestInfo_Ack;
   END_VAR

   VAR 
      Communication { S7_SetPoint := 'False'} : FB_OPC_SendReciveAck;
      staSource { ExternalAccessible := 'False'; ExternalVisible := 'False'; ExternalWritable := 'False'; S7_SetPoint := 'False'} : OPC_DestInfo;
      staAck { ExternalAccessible := 'False'; ExternalVisible := 'False'; ExternalWritable := 'False'; S7_SetPoint := 'False'} : OPC_DestInfo_Ack;
   END_VAR

   VAR_TEMP 
      Retval : Int;
   END_VAR


BEGIN
	// ==========================================================================================================================================
	// Company        : LogTech, s.r.o.
	// Created by     : Mahmoud Elnady
	// Block          : OPC_SendReciveAck
	// Project        : Lekarna, Chrudim -PLC001 -MCC001
	// Project number : 23-157
	// ==========================================================================================================================================
	
	
	//======================================================
	// Region: Communication Handling and Logging
	// Description: Manages the communication routine and logs
	//              events for message sending, acknowledgment
	//              reception, and acknowledgment timeout.
	//======================================================
	
	//------------------------------------------------------
	// Call communication routine
	//------------------------------------------------------
	REGION Communication routine
	    // Call communication routine
	    #Communication(SourceSeq := #staSource.SourceSeq,
	                   AckSeq := #staAck.AckSeq,
	                   Timeout := T#20s);
	END_REGION
	
	#Source.SourceSeq := #staSource.SourceSeq;
	#staAck.AckSeq := #Ack.AckSeq;
	
	
	//------------------------------------------------------
	// Log event when a new message is sent
	//------------------------------------------------------
	
	REGION Log event - new message
	    IF #Communication.Log.Send THEN
	        #Communication.Log.Send := FALSE;
	        // Logging
	        //(LOG)3003=$ Node $, new message sent, seq: $, palletID: $, WMSID: $
	        DB_LogMsg.LogMsg_7.Para_STRING_01.Data := #Source.DecisionPoint;
	        DB_LogMsg.LogMsg_7.Para_BYTE_02.Data := #Source.SourceSeq;
	        DB_LogMsg.LogMsg_7.Para_STRING_03.Data := #Source.Barcode;
	        DB_LogMsg.LogMsg_7.Para_STRING_04.Data := #Source.InformationPoint;
	        #Retval := FC_LogMsg(EventID := 3003, EventLevel := 2, EventGroup := 33, LogMsg := DB_LogMsg.LogMsg_7);
	    END_IF;
	END_REGION
	
	//------------------------------------------------------
	// Log event when new acknowledgment is received
	//------------------------------------------------------
	
	REGION Log event-New acknowledgment
	    IF #Communication.Log.New_Ack_received THEN
	        #Communication.Log.New_Ack_received := FALSE;
	        // Logging
	        //(LOG)3004=$ Node $, acknowledge received, seq: $, palletID: $, WMSID: $
	        DB_LogMsg.LogMsg_7.Para_BYTE_02.Data := #Ack.AckSeq;
	        #Retval := FC_LogMsg(EventID := 3004, EventLevel := 2, EventGroup := 33, LogMsg := DB_LogMsg.LogMsg_7);
	    END_IF;
	END_REGION
	
	//------------------------------------------------------
	// Log event when acknowledgment timeout occurs
	//------------------------------------------------------
	
	REGION Log event- acknowledgment timeout
	    IF #Communication.Log.Ack_timeout THEN
	        #Communication.Log.Ack_timeout := FALSE;
	        // Logging
	        //(LOG)3009=$ Node $, seq: $, acknowledge timeout!
	        DB_LogMsg.LogMsg_8.Para_STRING_01.Data := #Source.DecisionPoint;
	        DB_LogMsg.LogMsg_8.Para_BYTE_02.Data := #Communication.SendSeq;
	        #Retval := FC_LogMsg(EventID := 3009, EventLevel := 3, EventGroup := 33, LogMsg := DB_LogMsg.LogMsg_8);
	    END_IF;
	END_REGION
	
END_FUNCTION_BLOCK
END_NAMESPACE

NAMESPACE ProductionLine
FUNCTION_BLOCK FB_OPC_DestRequest
{ S7_Optimized_Access := 'TRUE' ; Published := 'FALSE' }
VERSION : 0.1
   VAR_IN_OUT 
      Source : OPC_DsetRequest;
      Ack : OPC_DestRequest_Ack;
   END_VAR

   VAR 
      Communication { S7_SetPoint := 'False'} : FB_OPC_SendReciveAck;
      staSource { ExternalAccessible := 'False'; ExternalVisible := 'False'; ExternalWritable := 'False'; S7_SetPoint := 'False'} : OPC_DsetRequest;
      staAck { ExternalAccessible := 'False'; ExternalVisible := 'False'; ExternalWritable := 'False'; S7_SetPoint := 'False'} : OPC_DestRequest_Ack;
   END_VAR

   VAR_TEMP 
      Retval : Int;
   END_VAR


BEGIN
	// ==========================================================================================================================================
	// Company        : LogTech, s.r.o.
	// Created by     : Mahmoud Elnady
	// Block          : OPC_SendReciveAck
	// Project        : Lekarna, Chrudim -PLC001 -MCC001
	// Project number : 23-157
	// ==========================================================================================================================================
	
	//======================================================
	// Region: Communication Handling and Logging
	// Description: Manages the communication routine and logs
	//              events for message sending, acknowledgment
	//              reception, and acknowledgment timeout.
	//======================================================
	
	//------------------------------------------------------
	// Call communication routine
	//------------------------------------------------------
	 REGION Communication Routine
	    // Call communication routine
	    #Communication(Timeout := T#15s,
	                   SourceSeq := #staSource.SourceSeq,
	                   AckSeq := #staAck.AckSeq);
	END_REGION 
	
	#Source.SourceSeq := #staSource.SourceSeq;
	#staAck.AckSeq := #Ack.AckSeq;
	
	//------------------------------------------------------
	// Log event when a new message is sent
	//------------------------------------------------------
	
	REGION Log event - new message
	    IF #Communication.Log.Send THEN
	        #Communication.Log.Send := FALSE;
	        // Logging
	        //(LOG)3001=$ Node $, new message sent, seq: $, palletID: $, WMSID $, barcode: $, weight: $, height: $, width: $, length: $, quality: $
	        DB_LogMsg.LogMsg_4.Para_STRING_01.Data := #Source.DecisionPoint;
	        DB_LogMsg.LogMsg_4.Para_BYTE_02.Data := #Source.SourceSeq;
	        //"DB_LogMsg".LogMsg_4.Para_STRING_03.Data := #Source.TotesID;
	        //"DB_LogMsg".LogMsg_4.Para_STRING_04.Data := #Source.WMSID;
	        DB_LogMsg.LogMsg_4.Para_STRING_05.Data := #Source.Barcode;
	        //"DB_LogMsg".LogMsg_4.Para_STRING_06.Data := #Source.Weight;
	               //"DB_LogMsg".LogMsg_4.Para_CHAR_09.Data := STRING_TO_CHAR(#Source.Length);
	        //"DB_LogMsg".LogMsg_4.Para_CHAR_10.Data := STRING_TO_CHAR(#Source.Quality);
	        
	        #Retval := FC_LogMsg(EventID := 3001,
	                               EventLevel := 2,
	                               EventGroup := 33,
	                               LogMsg := DB_LogMsg.LogMsg_4);
	    END_IF;
	END_REGION
	
	//------------------------------------------------------
	// Log event when new acknowledgment is received
	//------------------------------------------------------
	
	REGION Log event-New acknowledgment
	    IF #Communication.Log.New_Ack_received THEN
	        #Communication.Log.New_Ack_received := FALSE;
	        // Logging
	        //(LOG)3002=$ Node $, acknowledge received, seq: $, palletID: $, WMSID $, destination: $, no-stretch: $
	        DB_LogMsg.LogMsg_5.Para_STRING_01.Data := #Ack.DecisionPoint;
	        DB_LogMsg.LogMsg_5.Para_BYTE_02.Data := #Ack.AckSeq;
	        DB_LogMsg.LogMsg_5.Para_STRING_03.Data := #Ack.Barcode;
	        //"DB_LogMsg".LogMsg_5.Para_STRING_04.Data := #Ack.WMSID;
	        DB_LogMsg.LogMsg_5.Para_STRING_05.Data := #Ack.Destination;
	        
